xSuccess := __QUERYINTERFACE(iq_stExampleLeafModuleItf.i_ifDrive, ifRefActualValuesPosition);
IF NOT xSuccess OR ifRefActualValuesPosition = 0 THEN
	stExceptionModuleReaction1.etDiag		:= GD.ET_Diag.InputParameterInvalid;
	stExceptionModuleReaction1.udiDiagExt	:= ET_DiagExtExampleLeafModule.DriveInvalid;
	stExceptionModuleReaction1.sMsg			:= 'i_ifDrive : IF_RefActualValues not implemented.';
	
	ReportException(iq_stException := stExceptionModuleReaction1);		
END_IF
END_METHOD

METHOD SetOutputs
VAR_INPUT
END_VAR
IF xNotAbleToSetException THEN
	; (* Do nothing. Diag outputs show not reportable exception *)
	iq_stStandardModuleItf.q_xReady := FALSE;
ELSIF stModuleReaction.axReaction[TPL.ET_Reaction.AsyncStop] THEN
	iq_stStandardModuleItf.q_etDiag := GD.ET_Diag.ExecutionAborted;
	iq_stStandardModuleItf.q_udiDiagExt := ET_DiagExtExampleLeafModule.AsyncStop;
	iq_stStandardModuleItf.q_sDiagExt := 'AsyncStop';
	iq_stStandardModuleItf.q_sMsg := '';
	
	iq_stStandardModuleItf.q_xReady := FALSE;
ELSIF stModuleReaction.axReaction[TPL.ET_Reaction.SyncStopEL] THEN
	iq_stStandardModuleItf.q_etDiag := GD.ET_Diag.ExecutionAborted;
	iq_stStandardModuleItf.q_udiDiagExt := ET_DiagExtExampleLeafModule.SyncStopEL;
	iq_stStandardModuleItf.q_sDiagExt := 'SyncStopEL';
	iq_stStandardModuleItf.q_sMsg := '';
	
	iq_stStandardModuleItf.q_xReady := FALSE;
ELSIF stModuleReaction.axReaction[TPL.ET_Reaction.SyncStopEH] THEN
	iq_stStandardModuleItf.q_etDiag := GD.ET_Diag.ExecutionAborted;
	iq_stStandardModuleItf.q_udiDiagExt := ET_DiagExtExampleLeafModule.SyncStopEH;
	iq_stStandardModuleItf.q_sDiagExt := 'SyncStopEH';
	iq_stStandardModuleItf.q_sMsg := '';
	
	iq_stStandardModuleItf.q_xReady := FALSE;
ELSIF stModuleReaction.axReaction[TPL.ET_Reaction.StopEndOfCycle] THEN
	iq_stStandardModuleItf.q_etDiag := GD.ET_Diag.ExecutionAborted;
	iq_stStandardModuleItf.q_udiDiagExt := ET_DiagExtExampleLeafModule.StopEndOfCycle;
	iq_stStandardModuleItf.q_sDiagExt := 'StopEndOfCycle';
	iq_stStandardModuleItf.q_sMsg := '';
	
	iq_stStandardModuleItf.q_xReady := FALSE;
ELSE
	IF (iq_stExampleLeafModuleItf.q_etState <> ET_ExampleLeafModuleState.Disabled) AND
	   (iq_stExampleLeafModuleItf.q_etState <> ET_ExampleLeafModuleState.Initializing) THEN

		iq_stStandardModuleItf.q_xReady := TRUE;
	ELSE
		iq_stStandardModuleItf.q_xReady := FALSE;
	END_IF
		
	iq_stStandardModuleItf.q_etDiag := GD.ET_Diag.Ok;
	CASE iq_stExampleLeafModuleItf.q_etState OF
		ET_ExampleLeafModuleState.NoOp: 
			iq_stStandardModuleItf.q_udiDiagExt := ET_DiagExtExampleLeafModule.NoOp;
		ET_ExampleLeafModuleState.Disabled:
			iq_stStandardModuleItf.q_udiDiagExt := ET_DiagExtExampleLeafModule.Disabled;
		ET_ExampleLeafModuleState.Initializing:
			iq_stStandardModuleItf.q_udiDiagExt := ET_DiagExtExampleLeafModule.Initializing;
		ET_ExampleLeafModuleState.HomingWaitForStart:
			iq_stStandardModuleItf.q_udiDiagExt := ET_DiagExtExampleLeafModule.HomingWaitForStart;
		ET_ExampleLeafModuleState.HomingExecuting:
			iq_stStandardModuleItf.q_udiDiagExt := ET_DiagExtExampleLeafModule.HomingExecuting;
		ET_ExampleLeafModuleState.HomingDone:
			iq_stStandardModuleItf.q_udiDiagExt := ET_DiagExtExampleLeafModule.HomingDone;
		ET_ExampleLeafModuleState.AutoWaitForStart:
			iq_stStandardModuleItf.q_udiDiagExt := ET_DiagExtExampleLeafModule.AutoWaitForStart;
		ET_ExampleLeafModuleState.AutoRunning:
			iq_stStandardModuleItf.q_udiDiagExt := ET_DiagExtExampleLeafModule.AutoRunning;
	END_CASE
	iq_stStandardModuleItf.q_sDiagExt := FC_EtDiagExtExampleLeafModuleToString(i_etDiagExt := iq_stStandardModuleItf.q_udiDiagExt);
	iq_stStandardModuleItf.q_sMsg := '';
END_IF

IF fbLoggerPoint.etLogLevel >= APL.ET_LogLevel.StatusMessage THEN
	IF (iq_stExampleLeafModuleItf.q_etState <> etStateOld) THEN
		fbLoggerPoint.AddLogEntry(	i_etLogLevel	:= APL.ET_LogLevel.StatusMessage,
									i_etDiag		:= GD.ET_Diag.Ok,
									i_udiDiagExt	:= ET_DiagExtExampleLeafModule.Ok,
									i_sMessage		:= Standard.CONCAT('State changed to: ', FC_EtExampleLeafModuleStateToString(i_etState := iq_stExampleLeafModuleItf.q_etState)),
									q_etDiag		:= ,
									q_etDiagExt		:= );
	END_IF
	etStateOld := iq_stExampleLeafModuleItf.q_etState;
END_IF
END_METHOD

ACTION SignalSuccessfulExecution:
IF fbLoggerPoint.etLogLevel >= APL.ET_LogLevel.StatusMessage THEN
	fbLoggerPoint.AddLogEntry(	i_etLogLevel	:= APL.ET_LogLevel.StatusMessage,
								i_etDiag		:= GD.ET_Diag.Ok,
								i_udiDiagExt	:= ET_DiagExtExampleLeafModule.Ok,
								i_sMessage		:= Standard.CONCAT(Standard.CONCAT(Standard.CONCAT('Command done: ', FC_etExampleLeafModuleCmdToString(i_diCmd := iq_stStandardModuleItf.iq_diCmd)),' number: '),DINT_TO_STRING(iq_stStandardModuleItf.iq_diCmd)),
								q_etDiag		:= ,
								q_etDiagExt		:= );
END_IF

iq_stStandardModuleItf.q_xCMDActive := FALSE;
iq_stStandardModuleItf.q_xCMDDone := TRUE;
IF(iq_stStandardModuleItf.iq_diCMD = iq_stStandardModuleItf.q_diCMDActive) THEN
	iq_stStandardModuleItf.iq_diCMD := 0;
(* ELSE don't touch iq_diCMD *)
END_IF
END_ACTION

ACTION SignalUnSuccessfulExecution:
IF fbLoggerPoint.etLogLevel >= APL.ET_LogLevel.StatusMessage THEN
	fbLoggerPoint.AddLogEntry(	i_etLogLevel	:= APL.ET_LogLevel.StatusMessage,
								i_etDiag		:= GD.ET_Diag.Ok,
								i_udiDiagExt	:= ET_DiagExtExampleLeafModule.Ok,
								i_sMessage		:= Standard.CONCAT(Standard.CONCAT(Standard.CONCAT('Command failed: ', FC_etExampleLeafModuleCmdToString(i_diCmd := iq_stStandardModuleItf.iq_diCmd)),' number: '),DINT_TO_STRING(iq_stStandardModuleItf.iq_diCmd)),
								q_etDiag		:= ,
								q_etDiagExt		:= );
END_IF

iq_stStandardModuleItf.q_xCMDActive := FALSE;
iq_stStandardModuleItf.q_xCMDDone := FALSE;
IF(iq_stStandardModuleItf.iq_diCMD = iq_stStandardModuleItf.q_diCMDActive) THEN
	iq_stStandardModuleItf.iq_diCMD := - iq_stStandardModuleItf.iq_diCMD;
(* ELSE don't touch iq_diCMD *)
END_IF
END_ACTION

END_FUNCTION_BLOCK

// LMC_PacDrive/Application/TemplateFullProgrammingFramework/Examples/ExampleLeafModule/FC_EtExampleLeafModuleCmdToString
FUNCTION FC_EtExampleLeafModuleCmdToString : STRING[15]
VAR_INPUT
	i_diCmd		: DINT;
END_VAR
VAR_OUTPUT
	q_etDiag	: GD.ET_Diag := GD.ET_Diag.Ok;
	q_etDiagExt	: ET_DiagExtExampleLeafModule := ET_DiagExtExampleLeafModule.Ok;
END_VAR

CASE i_diCMD OF
	ET_ExampleLeafModuleCmd.Homing:
		FC_EtExampleLeafModuleCmdToString := 'Homing';
	ET_ExampleLeafModuleCmd.Auto:
		FC_EtExampleLeafModuleCmdToString := 'Auto';
	ET_ExampleLeafModuleCmd.Stop:
		FC_EtExampleLeafModuleCmdToString := 'Stop';
	ET_ExampleLeafModuleCmd.Start:
		FC_EtExampleLeafModuleCmdToString := 'Start';
	ET_ExampleLeafModuleCmd.Hold:
		FC_EtExampleLeafModuleCmdToString := 'Hold';
	ELSE
		FC_EtExampleLeafModuleCmdToString := CONCAT('Unkown Cmd ', DINT_TO_STRING(i_diCMD));
		
		q_etDiag := GD.ET_Diag.InputParameterInvalid;
		q_etDiagExt := ET_DiagExtExampleLeafModule.UnknownCmd;
END_CASE

END_FUNCTION

// LMC_PacDrive/Application/TemplateFullProgrammingFramework/Examples/ExampleLeafModule/FC_EtExampleLeafModuleStateToString
FUNCTION FC_EtExampleLeafModuleStateToString : STRING[25]
VAR_INPUT
	i_etState	: ET_ExampleLeafModuleState;
END_VAR
VAR_OUTPUT
	q_etDiag	: GD.ET_Diag := GD.ET_Diag.Ok;
	q_etDiagExt	: ET_DiagExtExampleLeafModule := ET_DiagExtExampleLeafModule.Ok;
END_VAR

CASE i_etState OF
	ET_ExampleLeafModuleState.Disabled:
		FC_EtExampleLeafModuleStateToString := 'Disabled';
	ET_ExampleLeafModuleState.Initializing:
		FC_EtExampleLeafModuleStateToString := 'Initializing';
	ET_ExampleLeafModuleState.NoOp:
		FC_EtExampleLeafModuleStateToString := 'NoOp';
	ET_ExampleLeafModuleState.HomingWaitForStart:
		FC_EtExampleLeafModuleStateToString := 'HomingWaitForStart';
	ET_ExampleLeafModuleState.HomingExecuting:
		FC_EtExampleLeafModuleStateToString := 'HomingExecuting';
	ET_ExampleLeafModuleState.HomingDone:
		FC_EtExampleLeafModuleStateToString := 'HomingDone';
	ET_ExampleLeafModuleState.AutoWaitForStart:
		FC_EtExampleLeafModuleStateToString := 'AutoWaitForStart';
	ET_ExampleLeafModuleState.AutoRunning:
		FC_EtExampleLeafModuleStateToString := 'AutoRunning';
	ELSE
		FC_EtExampleLeafModuleStateToString := CONCAT('Unkown State ', UDINT_TO_STRING(i_etState));
		
		q_etDiag := GD.ET_Diag.InputParameterInvalid;
		q_etDiagExt := ET_DiagExtExampleLeafModule.UnknownState;
END_CASE

END_FUNCTION

// LMC_PacDrive/Application/TemplateFullProgrammingFramework/Examples/ExampleLeafModule/FC_EtDiagExtExampleLeafModuleToString
FUNCTION FC_EtDiagExtExampleLeafModuleToString : STRING[80]

VAR_INPUT
	i_etDiagExt : ET_DiagExtExampleLeafModule;
END_VAR

VAR_OUTPUT
	q_etDiag	: GD.ET_Diag := GD.ET_Diag.Ok;
	q_etDiagExt	: ET_DiagExtExampleLeafModule := ET_DiagExtExampleLeafModule.Ok;
END_VAR

VAR
END_VAR

CASE i_etDiagExt OF
	ET_DiagExtExampleLeafModule.Ok:										FC_EtDiagExtExampleLeafModuleToString := 'Ok';
	ET_DiagExtExampleLeafModule.Disabled:								FC_EtDiagExtExampleLeafModuleToString := 'Disabled';
	ET_DiagExtExampleLeafModule.Initializing:							FC_EtDiagExtExampleLeafModuleToString := 'Initializing';
	ET_DiagExtExampleLeafModule.NoOp:									FC_EtDiagExtExampleLeafModuleToString := 'NoOp';
	ET_DiagExtExampleLeafModule.HomingWaitForStart:						FC_EtDiagExtExampleLeafModuleToString := 'HomingWaitForStart';
	ET_DiagExtExampleLeafModule.HomingExecuting:						FC_EtDiagExtExampleLeafModuleToString := 'HomingExecuting';
	ET_DiagExtExampleLeafModule.HomingDone:								FC_EtDiagExtExampleLeafModuleToString := 'HomingDone';
	ET_DiagExtExampleLeafModule.AutoWaitForStart:						FC_EtDiagExtExampleLeafModuleToString := 'AutoWaitForStart';
	ET_DiagExtExampleLeafModule.AutoRunning:							FC_EtDiagExtExampleLeafModuleToString := 'AutoRunning';
	ET_DiagExtExampleLeafModule.Working:								FC_EtDiagExtExampleLeafModuleToString := 'Working';

	ET_DiagExtExampleLeafModule.UnknownDiagExtExampleLeafModule:		FC_EtDiagExtExampleLeafModuleToString := 'UnknownDiagExtExampleLeafModule';
	ET_DiagExtExampleLeafModule.SubModuleAddInterfacesInvalidPointer:	FC_EtDiagExtExampleLeafModuleToString := 'SubModuleAddInterfacesInvalidPointer';
	ET_DiagExtExampleLeafModule.SubModuleConstantRange:					FC_EtDiagExtExampleLeafModuleToString := 'SubModuleConstantRange';
	ET_DiagExtExampleLeafModule.MissingExtInit:							FC_EtDiagExtExampleLeafModuleToString := 'MissingExtInit';
	ET_DiagExtExampleLeafModule.ReactionOffsetRange:					FC_EtDiagExtExampleLeafModuleToString := 'ReactionOffsetRange';
	ET_DiagExtExampleLeafModule.DriveInvalid:							FC_EtDiagExtExampleLeafModuleToString := 'DriveInvalid';
	
	ET_DiagExtExampleLeafModule.CmdUnknown:								FC_EtDiagExtExampleLeafModuleToString := 'CmdUnknown';
	ET_DiagExtExampleLeafModule.CmdImpossibleOverwrite:					FC_EtDiagExtExampleLeafModuleToString := 'CmdImpossibleOverwrite';
	ET_DiagExtExampleLeafModule.CmdImpossibleState:						FC_EtDiagExtExampleLeafModuleToString := 'CmdImpossibleState';
	ET_DiagExtExampleLeafModule.CmdImpossibleReaction:					FC_EtDiagExtExampleLeafModuleToString := 'CmdImpossibleReaction';
	
	ET_DiagExtExampleLeafModule.AsyncStop:								FC_EtDiagExtExampleLeafModuleToString := 'AsyncStop';
	ET_DiagExtExampleLeafModule.SyncStopEL:								FC_EtDiagExtExampleLeafModuleToString := 'SyncStopEL';
	ET_DiagExtExampleLeafModule.SyncStopEH:								FC_EtDiagExtExampleLeafModuleToString := 'SyncStopEH';
	ET_DiagExtExampleLeafModule.StopEndOfCycle:							FC_EtDiagExtExampleLeafModuleToString := 'StopEndOfCycle';
	
	ET_DiagExtExampleLeafModule.DriveFatalException:					FC_EtDiagExtExampleLeafModuleToString := 'DriveFatalException';
	ET_DiagExtExampleLeafModule.DriveException:							FC_EtDiagExtExampleLeafModuleToString := 'DriveException';
	ET_DiagExtExampleLeafModule.DriveWarning:							FC_EtDiagExtExampleLeafModuleToString := 'DriveWarning';
	
	ET_DiagExtExampleLeafModule.UnknownState:							FC_EtDiagExtExampleLeafModuleToString := 'UnknownState';
	ET_DiagExtExampleLeafModule.UnknownCmd:								FC_EtDiagExtExampleLeafModuleToString := 'UnknownCmd';
	ET_DiagExtExampleLeafModule.RandomException:						FC_EtDiagExtExampleLeafModuleToString := 'RandomException';

	ET_DiagExtExampleLeafModule.CurrentStandardItfInvalidPointer:		FC_EtDiagExtExampleLeafModuleToString := 'CurrentStandardItfInvalidPointer';
	ET_DiagExtExampleLeafModule.CurrentAddItfInvalidPointer:			FC_EtDiagExtExampleLeafModuleToString := 'CurrentAddItfInvalidPointer';
	
	ET_DiagExtExampleLeafModule.ParentInvalid:							FC_EtDiagExtExampleLeafModuleToString := 'ParentInvalid';
	ET_DiagExtExampleLeafModule.ParentNotRegistered:					FC_EtDiagExtExampleLeafModuleToString := 'ParentNotRegistered';
	ET_DiagExtExampleLeafModule.MaxNumberOfLoggerPointsExeeded:			FC_EtDiagExtExampleLeafModuleToString := 'MaxNumberOfLoggerPointsExeeded';
	ET_DiagExtExampleLeafModule.UnexpectedDiagExt:						FC_EtDiagExtExampleLeafModuleToString := 'UnexpectedDiagExt';
	
	ELSE
		FC_EtDiagExtExampleLeafModuleToString := Standard.CONCAT('Unkown ET_DiagExtExampleLeafModule ', UDINT_TO_STRING(i_etDiagExt));
		
		q_etDiag	:= GD.ET_Diag.InputParameterInvalid;
		q_etDiagExt	:= ET_DiagExtExampleLeafModule.UnknownDiagExtExampleLeafModule;
END_CASE

END_FUNCTION

// LMC_PacDrive/Application/TemplateFullProgrammingFramework/Examples/ExampleLeafModule/FB_ExampleLeafModuleController
FUNCTION_BLOCK FB_ExampleLeafModuleController

VAR_INPUT
	i_xEnable				: BOOL;
END_VAR

VAR_IN_OUT
	iq_stStandardModuleItf	: TPL.ST_StandardModuleInterface;
	iq_stStandardMotionItf	: TPL.ST_StandardMotionInterface;
	iq_stExceptionList		: TPL.ST_ExceptionList;
	iq_stLogDataList		: TPL.ST_LogDataList;
END_VAR

VAR_OUTPUT
	q_xActive				: BOOL;
	q_xReady				: BOOL;
	q_etDiag				: GD.ET_Diag := GD.ET_Diag.Ok;
	q_etDiagExt				: ET_DiagExtExampleLeafModule := ET_DiagExtExampleLeafModule.Disabled;
	q_sMsg					: STRING[80] := '';
END_VAR

VAR
	xEnableFlag				: BOOL;
	udiTmp					: UDINT;
END_VAR

IF i_xEnable AND NOT xEnableFlag THEN
	xEnableFlag	:= TRUE;
	
	q_xActive	:= TRUE;

	q_etDiag	:= GD.ET_Diag.Ok;
	q_etDiagExt := ET_DiagExtExampleLeafModule.Initializing;
	q_sMsg		:= '';
	
	IF ((iq_stStandardModuleItf.iq_stExt.udiNumberOfSubModules <> 0) AND 
	   ((iq_stStandardModuleItf.iq_stExt.pdwSubModulesAddItf = 0) OR (iq_stStandardModuleItf.iq_stExt.dwSubModulesItf = 0))) THEN
	   
		q_etDiag	:= GD.ET_Diag.ExecutionAborted;
		q_etDiagExt	:= ET_DiagExtExampleLeafModule.MissingExtInit;
		q_sMsg		:= 'Missing call of FC_UpdateExampleLeafModuleAddInterfaceStruct';

		RETURN;
	END_IF
	
	udiTmp := ET_ExceptionSource.ExampleLeafModule;
	
	q_xReady := TPL.FC_CheckSubModuleList(	i_dwModuleType		:= UDINT_TO_DWORD(ET_ModuleType.ExampleLeafModule),
											i_udiModuleId		:= iq_stStandardModuleItf.i_udiModuleId,
											i_sModuleName		:= iq_stStandardModuleItf.i_sModuleName,
											i_etSource			:= udiTmp (* Hack around compiler restrictions *),
											iq_stExt			:= iq_stStandardModuleItf.iq_stExt,
											iq_stExceptionList	:= iq_stExceptionList,
											iq_stLogDataList	:= iq_stLogDataList);
											
	IF NOT q_xReady THEN
		xEnableFlag := FALSE;
	END_IF

ELSIF NOT i_xEnable AND xEnableFlag THEN
	xEnableFlag	:= FALSE;
	
	(* No actions required, this simple module does not support jogging or any other things the XXXModuleController would have to handle *)
	q_xReady 	:= FALSE;
	q_xActive	:= FALSE;
	
	q_etDiag	:= GD.ET_Diag.Ok;
	q_etDiagExt	:= ET_DiagExtExampleLeafModule.Disabled;
	q_sMsg		:= '';
END_IF



IF q_xActive AND q_xReady THEN
	(* No actions required, this simple module does not support jogging or any other things the XXXModuleController would have to handle *)
	q_etDiag	:= GD.ET_Diag.Ok;
	q_etDiagExt := ET_DiagExtExampleLeafModule.Working;
	q_sMsg		:= '';
END_IF

END_FUNCTION_BLOCK

// LMC_PacDrive/Application/TemplateFullProgrammingFramework/Examples/ExampleLeafModule/FC_UpdateExampleLeafModuleAddInterfaceStruct
FUNCTION FC_UpdateExampleLeafModuleAddInterfaceStruct : BOOL

VAR_INPUT
	i_pdwSubModuleAddInterfaces		: POINTER TO DWORD;
	i_udiSubModuleConstant			: UDINT;
END_VAR

VAR_OUTPUT
	q_etDiag						: GD.ET_Diag := GD.ET_Diag.Ok;
	q_etDiagExt						: ET_DiagExtExampleLeafModule := ET_DiagExtExampleLeafModule.Ok;
	q_sMsg							: STRING[80] := '';
END_VAR

VAR_IN_OUT
	iq_stExampleLeafModuleInterface	: ST_ExampleLeafModuleInterface;
END_VAR

VAR
	pdwArrayPos						: POINTER TO DWORD;
END_VAR

IF i_pdwSubModuleAddInterfaces = 0 THEN
	q_etDiag	:= GD.ET_Diag.InputParameterInvalid;
	q_etDiagExt	:= ET_DiagExtExampleLeafModule.SubModuleAddInterfacesInvalidPointer;
	q_sMsg		:= '';
ELSIF i_udiSubModuleConstant < 1 THEN
	q_etDiag	:= GD.ET_Diag.InputParameterInvalid;
	q_etDiagExt := ET_DiagExtExampleLeafModule.SubModuleConstantRange;
	q_sMsg		:= '1 <= i_udiSubModuleConstant';
ELSE
	pdwArrayPos := i_pdwSubModuleAddInterfaces + UDINT_TO_DWORD((i_udiSubModuleConstant-1) * SIZEOF(pdwArrayPos^));
	pdwArrayPos^ := ADR(iq_stExampleLeafModuleInterface);
END_IF

END_FUNCTION

// LMC_PacDrive/Application/TemplateFullProgrammingFramework/EquipmentModules/MulticarrierModule/Multicarrier Stations/Test Multicarrier/FB_MotionTestStationBase
FUNCTION_BLOCK FB_MotionTestStationBase EXTENDS MCRS.FB_CoreStation 
VAR
	ifTargetStation 		: MCRS.IF_CoreStation;

	ifCarrier				 : MCR.IF_Carrier;

	etStationType 			  : ET_StationType;
	lrProcessPosInStation	  : LREAL;
	lrProcessGap			  : LREAL;

	lrMaxVelocity			: LREAL;
	lrMaxAcceleration		: LREAL;
	lrMaxDeceleration		: LREAL;
	lrMaxJerk				: LREAL;

	xError_loc				: BOOL;
	etResultSource_loc		: ET_ResultSource;
	udiEtResult_loc			: UDINT;
	sETResult_loc			: STRING(255);
	etResultStation_loc		: ET_ResultStation;
	etResultMCR_loc			: MCR.ET_Result;
	etResultMCRS_loc		: MCRS.ET_Result;
	sResultMsg_loc			: STRING(255);

	iState					: INT;
	xStationReadyForJob_loc	: BOOL;
	udiLoop					: UDINT;

	
END_VAR

END_FUNCTION_BLOCK

// LMC_PacDrive/Application/TemplateFullProgrammingFramework/Visualization/VIS_Main
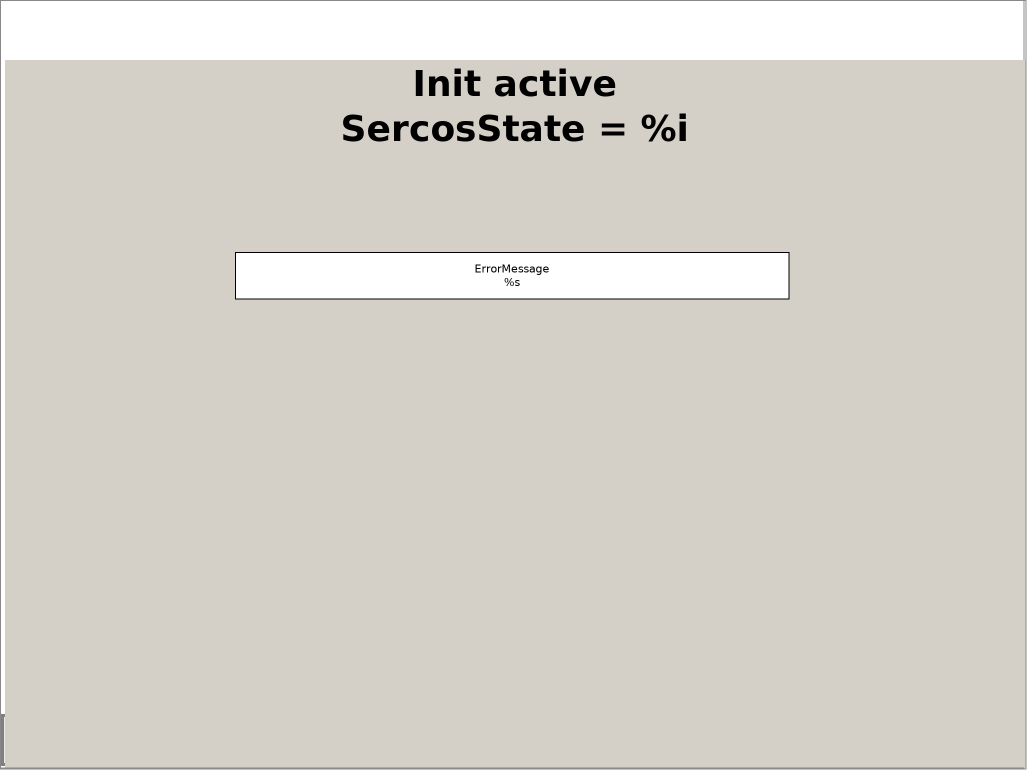
VISUALIZATION VIS_Main  // 1027x770
    Frame (0,0 1024x768)
        shows TPL.FR_NavControl1024x768(i_sTitle := 'Template: Main')
    Rectangle (105,63 688x480)
    Rectangle (105,63 688x40), "Machine - Control"
    Rectangle (105,102 688x78)
    Textfield (400,129 279x27)
    Button (693,119 90x44), "Diag Quit", colour toggle: SR_VisControl.vpq_xMachineInException
        p573394764: SR_VisControl.vpq_dwDiagQuitColor
        tap G_xDiagQuitEpas
    Textfield (117,129 279x27)
    Rectangle (402,130 275x25), "%s", text variable: SR_VisControl.vpq_etMainModuleControllerDiagExt, colour toggle: SR_VisControl.vpq_xMachineInException
        p2167032090: SR_VisControl.vpq_dwDiagQuitColor
    Rectangle (119,130 275x25), "%s", text variable: SR_VisControl.vpq_etMainModuleControllerDiag, colour toggle: SR_VisControl.vpq_xMachineInException
        p2167032090: SR_VisControl.vpq_dwDiagQuitColor
    Button (693,194 90x44), "Start", colour toggle: G_xStartEpas
        tap G_xStartEpas
    Button (693,253 90x44), "Stop", colour toggle: G_xStopEpas
        tap G_xStopEpas p3779583253=TRUE
    Button (693,312 90x44), "Jog +", colour toggle: G_xJogForwEpas
        tap G_xJogForwEpas p3779583253=TRUE
    Button (693,371 90x44), "Jog -", colour toggle: G_xJogBackEpas
        tap G_xJogBackEpas p3779583253=TRUE
    Button (125,195 90x44), "Prepare", colour toggle: G_xPrepareActive
        tap G_xDoPrepare
    Button (238,195 90x44), "Auto", colour toggle: G_xAutoActive
        tap G_xDoAuto
    Button (351,195 90x44), "Brake Release", colour toggle: G_xBrakeReleaseActive
        tap G_xDoBrakeRelease
    Button (464,195 90x44), "Jog Machine", colour toggle: G_xJogMachineActive
        tap G_xDoJogMachine
    Button (577,195 90x44), "Manual", colour toggle: G_xManualActive
        tap G_xDoManual
    Polyline (680,431) (793,431)
    Frame (693,442 90x90)
        shows TPL.FR_EmergencyStop90x90(i_xChangeColor := NOT G_xEmergencyEpas, i_xInvisible := FALSE, iq_xToggle := G_xEmergencyEpas)
    Frame (109,256 574x283)
        shows TPL.FR_ModuleCommandTable620x250(i_stCurrentModuleStandardItf := SR_VisControl.vpq_stMachineInterface, i_astActualCmdTable := SR_VisControl.vpq_astActualCmdTableMain, i_udiNumberOfCmdSteps := SR_VisControl.vpq_udiNumberOfCmdStepsMain, i_sCmdTitel := SR_VisControl.vpq_sCmdTitelMain, i_xDoEnable := SR_VisControl.vpq_xDoEnable, i_xDisableScrollUp := SR_VisControl.vpq_xDisableScrollUpMain, i_xDisableScrollDown := SR_VisControl.vpq_xDisableScrollDownMain, iq_udiIndexMin := SR_VisControl.vpiq_udiIndexMinMain)
        p2190627833: SR_VisControl.vpq_stMachineInterface
        p3492251336: SR_VisControl.vpq_stMachineInterface.iq_stExt.diActiveStep
    Frame (1,714 1024x54)
        shows FR_NavigationButtons()
    Rectangle (205,720 98x40), "Machine Control"
    Frame (821,60 200x430), invisible if: NOT SR_VisControl.vpiq_xShowControlFrame
        shows TPL.FR_MachineControl200x430(i_stMachineItf := SR_VisControl.vpq_stMachineInterface, i_xPrepareActive := G_xPrepareActive, i_xAutoActive := G_xAutoActive, i_xBrakeReleaseActive := G_xBrakeReleaseActive, i_xJogMachineActive := G_xJogMachineActive, i_xManualActive := G_xManualActive, i_xException := SR_VisControl.vpq_xMachineInException, i_dwDiagQuitColor := SR_VisControl.vpq_dwDiagQuitColor, iq_iPositionX := SR_VisControl.vpiq_iPositionX, iq_iPositionY := SR_VisControl.vpiq_iPositionY, iq_xEmergencyEpas := G_xEmergencyEpas, iq_xStartEpas := G_xStartEpas, iq_xStopEpas := G_xStopEpas, iq_xJogForwEpas := G_xJogForwEpas, iq_xJogBackEpas := G_xJogBackEpas, iq_xDoPrepare := G_xDoPrepare, iq_xDoAuto := G_xDoAuto, iq_xDoBrakeRelease := G_xDoBrakeRelease, iq_xDoJogMachine := G_xDoJogMachine, iq_xDoManual := G_xDoManual, iq_xDiagQuitEpas := G_xDiagQuitEpas)
        p1457045297: SR_VisControl.stMachineInterface.stQ.xError
        p1941967854: g_I_xEmergency_Epas
        p2531571229: g_I_xStart_Epas
        p1511842254: g_I_xStop_Epas
        p745511063: g_I_xJogForw_Epas
        p3518271027: g_I_xJogBack_Epas
        p1982879521: g_I_xErrorQuit_Epas
        p3866886353: SR_VisControl.dwErrorQuitColor
        p1761348311: SR_VisControl.vpq_stMachineInterface
        p3560616238: SR_VisControl.vpiq_iPositionX
        p2738717112: SR_VisControl.vpiq_iPositionY
    Rectangle (5,60 1020x707), "Init active SercosState = %i", text variable: G_ifSercos.State, invisible if: SR_MainMachine.xInitSuccessful
    Rectangle (235,252 554x47), "ErrorMessage %s", text variable: SR_MainMachine.stMachineInterface.q_sMsg, invisible if: SR_MainMachine.xInitSuccessful or not SR_MainMachine.xError
END_VISUALIZATION

// LMC_PacDrive/Application/TemplateFullProgrammingFramework/Visualization/Vis_Multicarrier
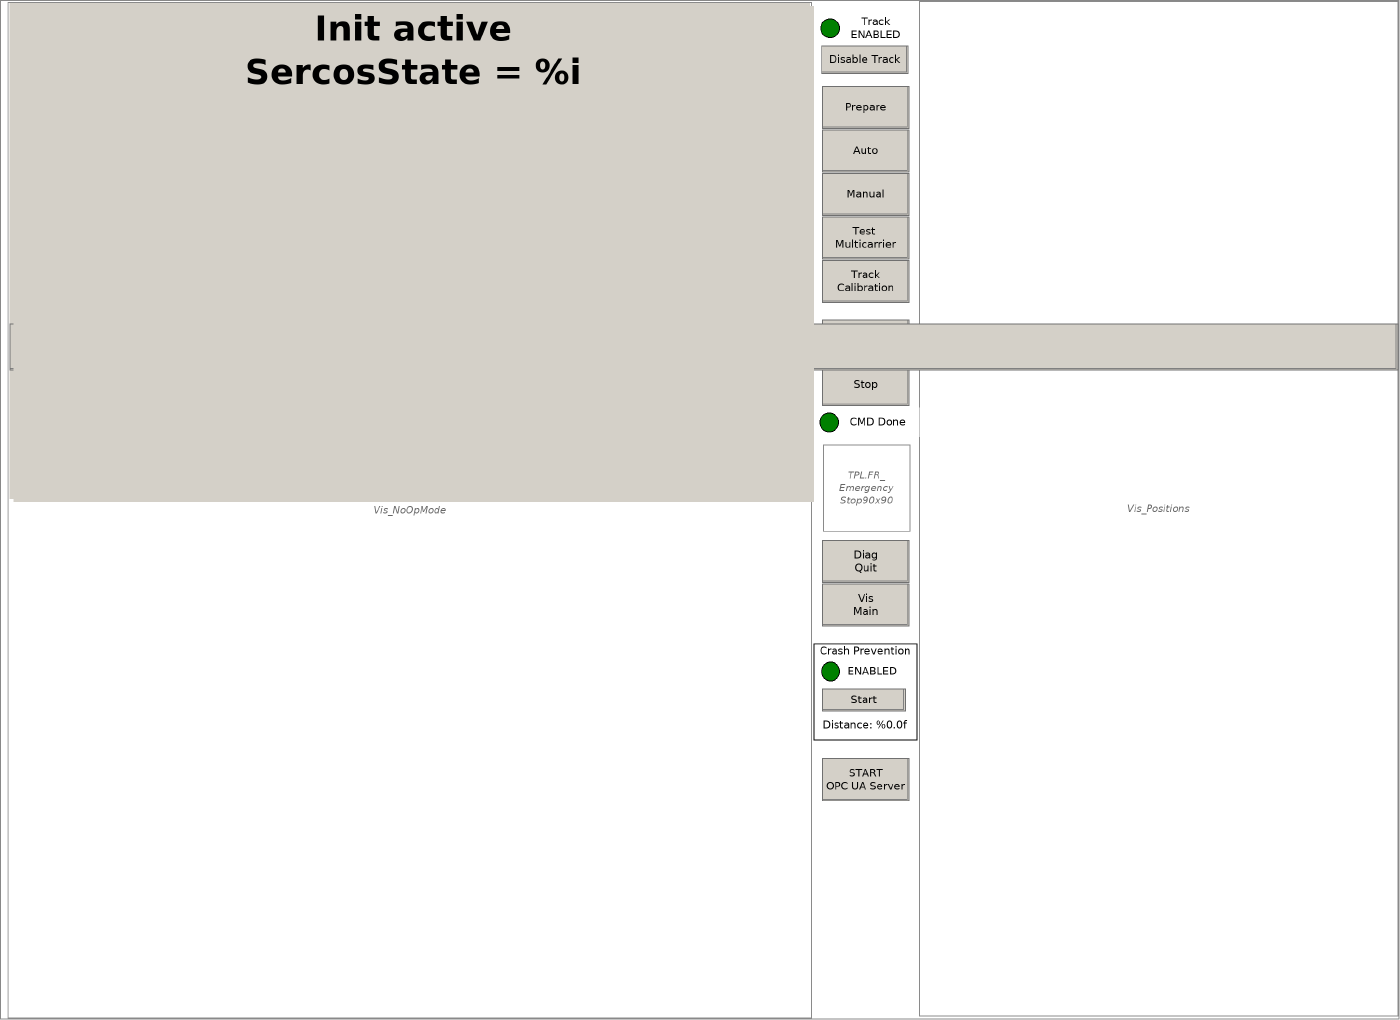
VISUALIZATION Vis_Multicarrier  // 1449x1056
    TabControl (8,2 832x1052), frame switch variable: SR_MultiCarrierModule.uiSetOpModeVis
        shows Vis_NoOpMode()
        shows Vis_Jogging()
        shows Vis_Auto()
        shows Vis_TestMulticarrier()
        shows Vis_TrackCalibration()
        [0]: TabTitle=None
        [1]: TabTitle=Manual
        [2]: TabTitle=Auto
        [3]: TabTitle=Test
        [4]: TabTitle=Trackcalibration
    TabControl (951,1 496x1051), frame switch variable: SR_MulticarrierModule.uiAdditionalVisTabs
        shows Vis_Positions()
        shows Vis_ApplicationLogger()
        shows Vis_Trace()
        shows Vis_Error()
        [0]: TabTitle=Positions
        [2]: TabTitle=Trace
        [3]: TabTitle=Error
    Frame (852,460 90x90)
        shows TPL.FR_EmergencyStop90x90(i_xChangeColor := NOT G_xEmergencyEpas, i_xInvisible := FALSE, iq_xToggle := G_xEmergencyEpas)
    Button (851,89 90x44), "Prepare", colour toggle: G_xPrepareActive
        tap G_xDoPrepare
    Button (851,559 90x44), "Diag Quit", colour toggle: SR_VisControl.vpq_xMachineInException
        p573394764: SR_VisControl.vpq_dwDiagQuitColor
        tap G_xDiagQuitEpas
    Button (851,134 90x44), "Auto", colour toggle: G_xAutoActive
        tap G_xDoAuto
    Button (851,179 90x44), "Manual", colour toggle: G_xManualActive
        tap G_xDoManual
    Button (851,224 90x44), "Test Multicarrier", colour toggle: G_xTestMulticarrierActive
        tap G_xDoTestMulticarrier
    Button (851,331 90x44), "Start", colour toggle: G_xStartEpas
        tap G_xStartEpas
    Button (851,376 90x44), "Stop", colour toggle: G_xStopEpas
        tap G_xStopEpas p3779583253=TRUE
    Button (851,785 90x44), "START OPC UA Server", colour toggle: SR_OpcUa.xStartUaServer
        toggle SR_OpcUa.xStartUaServer
    Group (848,422 103x30)
        Rectangle (18,0 85x30), "CMD Done"
        Ellipse (0,5 20x20), colour toggle: SR_MainMachine.fbModuleController.q_xCmdDone
    Rectangle (864,14 85x30), "Track ENABLED"
    Ellipse (849,19 20x20), colour toggle: SR_MultiCarrierModule.xEnableTrackSuccessful
    Button (850,47 90x29), "Enable Track", colour toggle: SR_MultiCarrierModule.xControlEnable, invisible if: SR_MultiCarrierModule.iStateOpMode > 0 or SR_MultiCarrierModule.xControlEnable
        toggle SR_MultiCarrierModule.xControlEnable
    Button (850,47 90x29), "Disable Track", invisible if: SR_MultiCarrierModule.iStateOpMode > 0 or not SR_MultiCarrierModule.xControlEnable
        toggle SR_MultiCarrierModule.xControlEnable
    Button (851,604 90x44), "Vis Main"
        OnMouseClick:  Assign=VIS_Main, Type=Assignment
    Rectangle (842,666 107x100), "Crash Prevention"
    Button (851,713 86x23), "Start", colour toggle: SR_MultiCarrierModule.xStartFbCrashPrevention
        toggle SR_MultiCarrierModule.xStartFbCrashPrevention
    Rectangle (863,680 80x30), "ENABLED"
    Ellipse (850,685 19x20), colour toggle: SR_MultiCarrierModule.xActiveFbCrashPrevention
    Rectangle (847,737 96x27), "Distance: %0.0f", tooltip "min distance between two Carriers (rear- and front offset under consideration)", text variable: GVL_Project.G_lrCrashDistance
        OnMouseClick: write the text variable via Default, min 0
    Rectangle (10,3 828x513), "Prepare Mode active", invisible if: SR_MulticarrierModule.iStateOpMode < 200 or SR_MulticarrierModule.iStateOpMode > 260
    Rectangle (149,192 554x47), "ErrorMessage %s", text variable: SR_MainMachine.stMachineInterface.q_sMsg, invisible if: SR_MainMachine.xInitSuccessful or not SR_MainMachine.xError
    Button (10,335 1437x48), "Enable Vis", colour toggle: G_xDoEnableVis, invisible if: G_xDoEnableVis
        toggle G_xDoEnableVis
    Rectangle (14,6 828x513), "Init active SercosState = %i", text variable: G_ifSercos.State, invisible if: SR_MainMachine.xInitSuccessful
    Button (851,269 90x44), "Track Calibration", colour toggle: G_xTrackCalibrationActive, invisible if: GVL_Project.Gc_xTrackCalibrationOfMulticarrier = false
        tap G_xDoTrackCalibration
END_VISUALIZATION

// LMC_PacDrive/Application/TemplateFullProgrammingFramework/Visualization/Examples/FR_ButtonAssignId
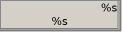
VISUALIZATION FR_ButtonAssignId  // 122x32
VAR_INPUT
	i_udiId : UDINT;
	i_sName : STRING[80];
	i_udiCurrentModuleId : UDINT;
END_VAR
VAR_IN_OUT
	iq_udiAssignTarget : UDINT;
END_VAR
    Button (0,0 120x30), "%s", text variable: i_sName, colour toggle: i_udiId = i_udiCurrentModuleId, invisible if: i_udiId<1
    Rectangle (0,0 119x29), "%s", text variable: i_udiId, invisible if: i_udiId<1
        OnMouseUp: execute { iq_udiAssignTarget := i_udiId; }
END_VISUALIZATION

// LMC_PacDrive/Application/TemplateFullProgrammingFramework/Visualization/Examples/FR_ExampleLeafModule
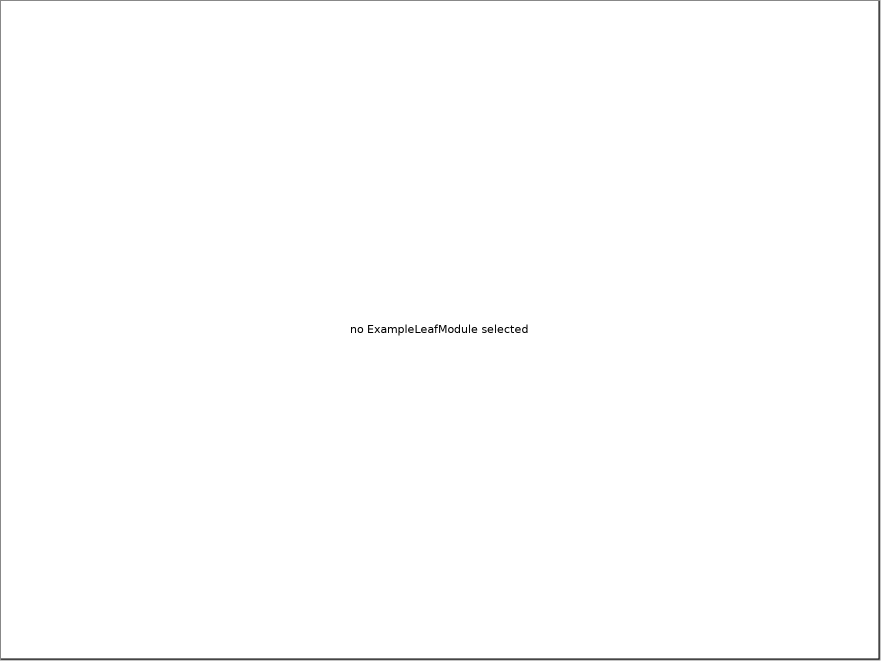
VISUALIZATION FR_ExampleLeafModule  // 881x661
VAR_IN_OUT
	iq_xModuleReactionDown				: BOOL;
	iq_xModuleReactionUp				: BOOL;
	iq_diStartStepToSet					: DINT;
	iq_diCmdToSet						: DINT;
	iq_xEnableModuleClicked				: BOOL;
	iq_xSetCmdClicked					: BOOL;
	iq_fbVisContExHandling				: TPL.FB_VisControllerExceptionHandling;
	iq_fbExampleLeafModuleVisController : FB_ExampleLeafModuleVisController;
END_VAR
VAR_INPUT
	i_stCurrentModuleStandardInterface : TPL.ST_StandardModuleInterface;
	i_sCurrentModuleReaction	: STRING[80];
	i_udiModuleReactionIndexMin : UDINT;
	i_axModuleReaction			: ARRAY [1..10] OF BOOL;
	i_udiNumberOfReactions 		: UDINT;
END_VAR
    Frame (0,0 380x211)
        shows TPL.FR_StandardModuleInterface380x220(i_stCurrentModuleStandardItf := i_stCurrentModuleStandardInterface, i_sCurrentModuleReaction := i_sCurrentModuleReaction, i_udiModuleReactionIndexMin := i_udiModuleReactionIndexMin, i_axModuleReaction := i_axModuleReaction, i_udiNumberOfReactions := i_udiNumberOfReactions, iq_xModuleReactionDown := iq_xModuleReactionDown, iq_xModuleReactionUp := iq_xModuleReactionUp, iq_diStartStepToSet := iq_diStartStepToSet, iq_diCmdToSet := iq_diCmdToSet, iq_xEnableModuleClicked := iq_xEnableModuleClicked, iq_xSetCmdClicked := iq_xSetCmdClicked, iq_fbVisContExHandling := iq_fbVisContExHandling)
        p3339340907: i_sZoomToVisModuleErrors
        p1094400588: i_xCurrentIsOfMyType
        p1029787830: i_fbVisContExHandling
        p2258115317: i_iModuleErrorReactionIndexMin
        p2777435286: i_axModuleErrorReaction
        p214250784: i_diNumberOfErrorreactions
        p311732222: iq_stCurrentModuleStandardInterface
        p640132070: iq_xModuleErrorReactionDown
        p4234372197: iq_xModuleErrorReactionUp
        p2938682392: iq_xEnableModule_Clicked
        p3592490199: iq_xSetCmd_Clicked
        p2307280719: iq_stCurrentModuleStandardInterface
        p2190627833: i_stCurrentModuleStandardInterface
    Rectangle (0,0 879x659), "no ExampleLeafModule selected", invisible if: iq_fbExampleLeafModuleVisController.xCurrentIsOfMyType
END_VISUALIZATION

// LMC_PacDrive/Application/TemplateFullProgrammingFramework/Visualization/Examples/FR_ExampleLeafModuleSelect
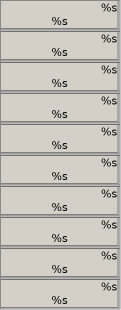
VISUALIZATION FR_ExampleLeafModuleSelect  // 121x310
VAR_IN_OUT
	iq_fbExampleLeafModuleVisController : FB_ExampleLeafModuleVisController;
END_VAR
VAR_INPUT
	i_stCurrentModuleStandardInterface : TPL.ST_StandardModuleInterface;
END_VAR
    Frame (0,0 119x29)
        shows FR_ButtonAssignId(i_udiId := iq_fbExampleLeafModuleVisController.audiExampleLeafModuleId[1], i_sName := iq_fbExampleLeafModuleVisController.asExampleLeafModuleName[1], i_udiCurrentModuleId := i_stCurrentModuleStandardInterface.i_udiModuleId, iq_udiAssignTarget := iq_fbExampleLeafModuleVisController.udiSetAsCurrentModule)
    Frame (0,31 119x29)
        shows FR_ButtonAssignId(i_udiId := iq_fbExampleLeafModuleVisController.audiExampleLeafModuleId[2], i_sName := iq_fbExampleLeafModuleVisController.asExampleLeafModuleName[2], i_udiCurrentModuleId := i_stCurrentModuleStandardInterface.i_udiModuleId, iq_udiAssignTarget := iq_fbExampleLeafModuleVisController.udiSetAsCurrentModule)
    Frame (0,62 119x29)
        shows FR_ButtonAssignId(i_udiId := iq_fbExampleLeafModuleVisController.audiExampleLeafModuleId[3], i_sName := iq_fbExampleLeafModuleVisController.asExampleLeafModuleName[3], i_udiCurrentModuleId := i_stCurrentModuleStandardInterface.i_udiModuleId, iq_udiAssignTarget := iq_fbExampleLeafModuleVisController.udiSetAsCurrentModule)
    Frame (0,93 119x29)
        shows FR_ButtonAssignId(i_udiId := iq_fbExampleLeafModuleVisController.audiExampleLeafModuleId[4], i_sName := iq_fbExampleLeafModuleVisController.asExampleLeafModuleName[4], i_udiCurrentModuleId := i_stCurrentModuleStandardInterface.i_udiModuleId, iq_udiAssignTarget := iq_fbExampleLeafModuleVisController.udiSetAsCurrentModule)
    Frame (0,124 119x29)
        shows FR_ButtonAssignId(i_udiId := iq_fbExampleLeafModuleVisController.audiExampleLeafModuleId[5], i_sName := iq_fbExampleLeafModuleVisController.asExampleLeafModuleName[5], i_udiCurrentModuleId := i_stCurrentModuleStandardInterface.i_udiModuleId, iq_udiAssignTarget := iq_fbExampleLeafModuleVisController.udiSetAsCurrentModule)
    Frame (0,155 119x29)
        shows FR_ButtonAssignId(i_udiId := iq_fbExampleLeafModuleVisController.audiExampleLeafModuleId[6], i_sName := iq_fbExampleLeafModuleVisController.asExampleLeafModuleName[6], i_udiCurrentModuleId := i_stCurrentModuleStandardInterface.i_udiModuleId, iq_udiAssignTarget := iq_fbExampleLeafModuleVisController.udiSetAsCurrentModule)
    Frame (0,186 119x29)
        shows FR_ButtonAssignId(i_udiId := iq_fbExampleLeafModuleVisController.audiExampleLeafModuleId[7], i_sName := iq_fbExampleLeafModuleVisController.asExampleLeafModuleName[7], i_udiCurrentModuleId := i_stCurrentModuleStandardInterface.i_udiModuleId, iq_udiAssignTarget := iq_fbExampleLeafModuleVisController.udiSetAsCurrentModule)
    Frame (0,217 119x29)
        shows FR_ButtonAssignId(i_udiId := iq_fbExampleLeafModuleVisController.audiExampleLeafModuleId[8], i_sName := iq_fbExampleLeafModuleVisController.asExampleLeafModuleName[8], i_udiCurrentModuleId := i_stCurrentModuleStandardInterface.i_udiModuleId, iq_udiAssignTarget := iq_fbExampleLeafModuleVisController.udiSetAsCurrentModule)
    Frame (0,248 119x29)
        shows FR_ButtonAssignId(i_udiId := iq_fbExampleLeafModuleVisController.audiExampleLeafModuleId[9], i_sName := iq_fbExampleLeafModuleVisController.asExampleLeafModuleName[9], i_udiCurrentModuleId := i_stCurrentModuleStandardInterface.i_udiModuleId, iq_udiAssignTarget := iq_fbExampleLeafModuleVisController.udiSetAsCurrentModule)
    Frame (0,279 119x29)
        shows FR_ButtonAssignId(i_udiId := iq_fbExampleLeafModuleVisController.audiExampleLeafModuleId[10], i_sName := iq_fbExampleLeafModuleVisController.asExampleLeafModuleName[10], i_udiCurrentModuleId := i_stCurrentModuleStandardInterface.i_udiModuleId, iq_udiAssignTarget := iq_fbExampleLeafModuleVisController.udiSetAsCurrentModule)
END_VISUALIZATION

// LMC_PacDrive/Application/TemplateFullProgrammingFramework/Visualization/Examples/VIS_ExampleLeafModule
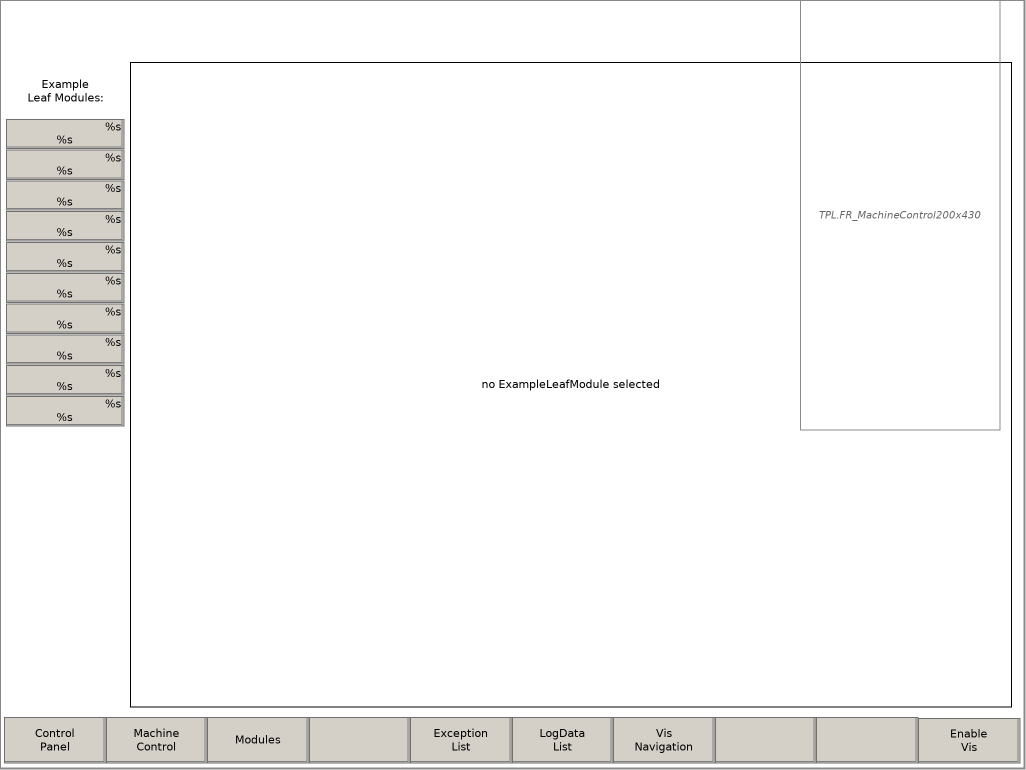
VISUALIZATION VIS_ExampleLeafModule  // 1026x770
    Frame (0,0 1024x768)
        shows TPL.FR_Nav1024x768(i_sTitle := 'Example Leaf Module')
    Frame (6,119 119x308)
        shows FR_ExampleLeafModuleSelect(i_stCurrentModuleStandardInterface := SR_VisControl.vpq_stCurrentModuleStandardInterface, iq_fbExampleLeafModuleVisController := SR_VisControl.vpiq_fbExampleLeafModuleVisController)
    Rectangle (6,65 119x52), "Example Leaf Modules:"
    Frame (130,62 884x647)
        shows FR_ExampleLeafModule(i_stCurrentModuleStandardInterface := SR_VisControl.vpq_stCurrentModuleStandardInterface, i_sCurrentModuleReaction := SR_VisControl.vpq_sCurrentModuleReaction, i_udiModuleReactionIndexMin := SR_VisControl.vpq_udiModuleReactionIndexMin, i_axModuleReaction := SR_VisControl.vpq_axModuleReaction, i_udiNumberOfReactions := TPL.Gc_udiMaxNumberOfReactions, iq_xModuleReactionDown := SR_VisControl.vpiq_xModuleReactionDown, iq_xModuleReactionUp := SR_VisControl.vpiq_xModuleReactionUp, iq_diStartStepToSet := SR_VisControl.vpiq_diStartStepToSet, iq_diCmdToSet := SR_VisControl.vpiq_diCmdToSet, iq_xEnableModuleClicked := SR_VisControl.vpiq_xEnableModuleClicked, iq_xSetCmdClicked := SR_VisControl.vpiq_xSetCmdClicked, iq_fbVisContExHandling := SR_VisControl.vpiq_fbVisContExHandling, iq_fbExampleLeafModuleVisController := SR_VisControl.vpiq_fbExampleLeafModuleVisController)
    Button (4,717 102x46), "Control Panel", colour toggle: SR_VisControl.vpiq_xShowControlFrame
        toggle SR_VisControl.vpiq_xShowControlFrame
    Button (106,717 101x46), "Machine Control"
        OnMouseClick:  Assign=VIS_Main, Type=Assignment
    Button (207,717 102x46), "Modules"
        OnMouseClick:  Assign=VIS_Modules, Type=Assignment
    Button (309,717 101x46)
    Button (410,717 102x46), "Exception List"
        OnMouseClick:  Assign=VIS_ExceptionList, Type=Assignment
    Button (512,717 101x46), "LogData List"
        OnMouseClick:  Assign=VIS_LogDataList, Type=Assignment
    Button (613,717 102x46), "Vis Navigation"
        OnMouseClick:  Assign=VIS_VisNavigation, Type=Assignment
    Button (715,717 101x46)
    Button (816,717 102x46)
    Button (918,718 102x45), "Enable Vis", colour toggle: G_xDoEnableVis
        OnMouseClick:  ToggleVariable=G_xDoEnableVis
    Frame (800,0 200x430), invisible if: NOT SR_VisControl.vpiq_xShowControlFrame
        shows TPL.FR_MachineControl200x430(i_stMachineItf := SR_VisControl.vpq_stMachineInterface, i_xPrepareActive := G_xPrepareActive, i_xAutoActive := G_xAutoActive, i_xBrakeReleaseActive := G_xBrakeReleaseActive, i_xJogMachineActive := G_xJogMachineActive, i_xManualActive := G_xManualActive, i_xException := SR_VisControl.vpq_xMachineInException, i_dwDiagQuitColor := SR_VisControl.vpq_dwDiagQuitColor, iq_iPositionX := SR_VisControl.vpiq_iPositionX, iq_iPositionY := SR_VisControl.vpiq_iPositionY, iq_xEmergencyEpas := G_xEmergencyEpas, iq_xStartEpas := G_xStartEpas, iq_xStopEpas := G_xStopEpas, iq_xJogForwEpas := G_xJogForwEpas, iq_xJogBackEpas := G_xJogBackEpas, iq_xDoPrepare := G_xDoPrepare, iq_xDoAuto := G_xDoAuto, iq_xDoBrakeRelease := G_xDoBrakeRelease, iq_xDoJogMachine := G_xDoJogMachine, iq_xDoManual := G_xDoManual, iq_xDiagQuitEpas := G_xDiagQuitEpas)
        p1457045297: SR_VisControl.stMachineInterface.stQ.xError
        p1941967854: g_I_xEmergency_Epas
        p2531571229: g_I_xStart_Epas
        p1511842254: g_I_xStop_Epas
        p745511063: g_I_xJogForw_Epas
        p3518271027: g_I_xJogBack_Epas
        p1982879521: g_I_xErrorQuit_Epas
        p3866886353: SR_VisControl.dwErrorQuitColor
        p1761348311: SR_VisControl.vpq_stMachineInterface
        p3560616238: SR_VisControl.vpiq_iPositionX - 800
        p2738717112: SR_VisControl.vpiq_iPositionY
END_VISUALIZATION

// LMC_PacDrive/Application/TemplateFullProgrammingFramework/Visualization/FramesProject/FR_ControlModuleTypes
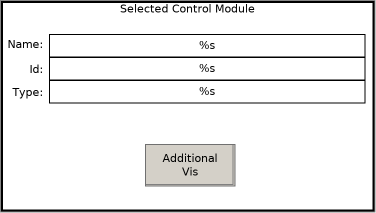
VISUALIZATION FR_ControlModuleTypes  // 376x213
VAR_INPUT
	i_sControlModuleName		: STRING[80];
	i_diControlModuleNumber		: DINT;
	i_diControlModuleType		: DINT;
END_VAR
    Rectangle (1,1 373x210), "Selected Control Module"
    Button (145,144 90x42), "Additional Vis"
        OnMouseClick:  AssignExpr=i_sZoomToControlModuleVis, Assign=VIS_ControlModule, Type=Assignment
    Textfield (49,34 316x23), "%s", text variable: i_sControlModuleName
    Rectangle (7,36 39x17), "Name:"
    Textfield (49,57 316x23), "%s", text variable: i_diControlModuleNumber
    Rectangle (7,61 39x17), "Id:"
    Rectangle (7,84 39x17), "Type:"
    Textfield (49,80 316x23), "%s", text variable: i_diControlModuleType
END_VISUALIZATION

// LMC_PacDrive/Application/TemplateFullProgrammingFramework/Visualization/FramesProject/FR_NavigationButtons
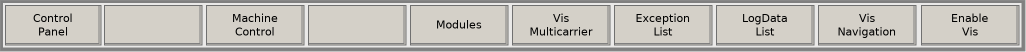
VISUALIZATION FR_NavigationButtons  // 1026x52
    Rectangle (0,0 1024x50)
    Button (410,5 98x40), "Modules"
        OnMouseClick:  Assign=VIS_Modules, Type=Assignment
    Button (5,5 96x40), "Control Panel", colour toggle: SR_VisControl.vpiq_xShowControlFrame
        toggle SR_VisControl.vpiq_xShowControlFrame
    Button (614,5 98x40), "Exception List"
        OnMouseClick:  Assign=VIS_ExceptionList, Type=Assignment
    Button (716,5 98x40), "LogData List"
        OnMouseClick:  Assign=VIS_LogDataList, Type=Assignment
    Button (818,5 98x40), "Vis Navigation"
        OnMouseClick:  Assign=VIS_VisNavigation, Type=Assignment
    Button (308,5 98x40)
    Button (104,5 98x40)
    Button (206,5 98x40), "Machine Control"
        OnMouseClick:  Assign=VIS_Main, Type=Assignment
    Button (921,5 98x40), "Enable Vis", colour toggle: G_xDoEnableVis
        toggle G_xDoEnableVis
    Button (512,5 98x40), "Vis Multicarrier"
        OnMouseDown:  Assign=Vis_Multicarrier, Type=Assignment
END_VISUALIZATION

// LMC_PacDrive/Application/TemplateFullProgrammingFramework/Visualization/FramesProject/FR_OtherModuleTypes
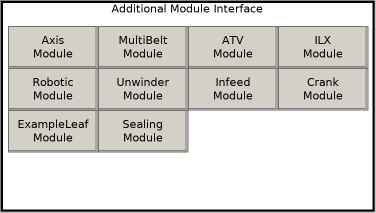
VISUALIZATION FR_OtherModuleTypes  // 376x213
    Rectangle (1,1 373x210), "Additional Module Interface"
    Button (8,26 90x42), "Axis Module", invisible if: SR_VisControl.vpq_stCurrentModuleStandardInterface.q_dwModuleType <> 3
        OnMouseClick:  Assign=VIS_AxisModule, Type=Assignment
    Button (98,26 90x42), "MultiBelt Module", invisible if: SR_VisControl.vpq_stCurrentModuleStandardInterface.q_dwModuleType <> 4
    Button (188,26 90x42), "ATV Module", invisible if: SR_VisControl.vpq_stCurrentModuleStandardInterface.q_dwModuleType <> 9
    Button (278,26 90x42), "ILX Module", invisible if: SR_VisControl.vpq_stCurrentModuleStandardInterface.q_dwModuleType <> 10
    Button (8,68 90x42), "Robotic Module", invisible if: SR_VisControl.vpq_stCurrentModuleStandardInterface.q_dwModuleType <> 6
    Button (8,110 90x42), "ExampleLeaf Module", invisible if: SR_VisControl.vpq_stCurrentModuleStandardInterface.q_dwModuleType <> 15000
        OnMouseClick:  AssignExpr=i_sZoomToExampleLeafModule, Assign=VIS_ExampleLeafModules, Type=Assignment
    Button (98,68 90x42), "Unwinder Module", invisible if: SR_VisControl.vpq_stCurrentModuleStandardInterface.q_dwModuleType <> 7
    Button (188,68 90x42), "Infeed Module", invisible if: SR_VisControl.vpq_stCurrentModuleStandardInterface.q_dwModuleType <> 5
    Button (278,68 90x42), "Crank Module", invisible if: SR_VisControl.vpq_stCurrentModuleStandardInterface.q_dwModuleType <> 11
    Button (98,110 90x42), "Sealing Module", invisible if: SR_VisControl.vpq_stCurrentModuleStandardInterface.q_dwModuleType <> 8
END_VISUALIZATION

// LMC_PacDrive/Application/TemplateFullProgrammingFramework/Visualization/Multicarrier/FR_CarDist
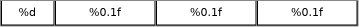
VISUALIZATION FR_CarDist  // 359x27
VAR_IN_OUT
	i_ifCarrierFeedback : MCR.IF_CarrierFeedback;
END_VAR
    Rectangle (1,0 53x25), "%d", text variable: i_ifCarrierFeedback.udiCarrierIndex
    Rectangle (55,0 100x25), "%0.1f", text variable: i_ifCarrierFeedback.ifFeedbackMotionValues.lrRefPosition
    Rectangle (156,0 100x25), "%0.1f", text variable: i_ifCarrierFeedback.ifFeedbackMotionValues.lrRefPosition
    Rectangle (257,0 100x25), "%0.1f", text variable: i_ifCarrierFeedback.ifFeedbackMotionValues.lrRefPosition
    Rectangle (55,0 100x25), "%0.1f", text variable: i_ifCarrierFeedback.ifFeedbackMotionValues.lrRefTrackPosition, invisible if: SR_MulticarrierModule.etVisPosColumn1 <> ET_VisPosGapDist.RefTrackPosition
    Rectangle (55,0 100x25), "%0.1f", text variable: i_ifCarrierFeedback.ifFeedbackToInFront.lrGapToCarrierInFront, invisible if: SR_MulticarrierModule.etVisPosColumn1 <> ET_VisPosGapDist.GapToCarrierInFront
    Rectangle (55,0 100x25), "%0.1f", text variable: i_ifCarrierFeedback.ifFeedbackToInFront.lrDistanceToCarrierInFront, invisible if: SR_MulticarrierModule.etVisPosColumn1 <> ET_VisPosGapDist.DistanceToCarrierInFront
    Rectangle (55,0 100x25), "%0.1f", text variable: i_ifCarrierFeedback.ifFeedbackToBehind.lrGapToCarrierBehind, invisible if: SR_MulticarrierModule.etVisPosColumn1 <> ET_VisPosGapDist.GapToCarrierBehind
    Rectangle (55,0 100x25), "%0.1f", text variable: i_ifCarrierFeedback.ifFeedbackToBehind.lrDistanceToCarrierBehind, invisible if: SR_MulticarrierModule.etVisPosColumn1 <> ET_VisPosGapDist.DistanceToCarrierBehind
    Rectangle (156,0 100x25), "%0.1f", text variable: i_ifCarrierFeedback.ifFeedbackMotionValues.lrRefTrackPosition, invisible if: SR_MulticarrierModule.etVisPosColumn2 <> ET_VisPosGapDist.RefTrackPosition
    Rectangle (156,0 100x25), "%0.1f", text variable: i_ifCarrierFeedback.ifFeedbackToInFront.lrGapToCarrierInFront, invisible if: SR_MulticarrierModule.etVisPosColumn2 <> ET_VisPosGapDist.GapToCarrierInFront
    Rectangle (156,0 100x25), "%0.1f", text variable: i_ifCarrierFeedback.ifFeedbackToInFront.lrDistanceToCarrierInFront, invisible if: SR_MulticarrierModule.etVisPosColumn2 <> ET_VisPosGapDist.DistanceToCarrierInFront
    Rectangle (156,0 100x25), "%0.1f", text variable: i_ifCarrierFeedback.ifFeedbackToBehind.lrGapToCarrierBehind, invisible if: SR_MulticarrierModule.etVisPosColumn2 <> ET_VisPosGapDist.GapToCarrierBehind
    Rectangle (156,0 100x25), "%0.1f", text variable: i_ifCarrierFeedback.ifFeedbackToBehind.lrDistanceToCarrierBehind, invisible if: SR_MulticarrierModule.etVisPosColumn2 <> ET_VisPosGapDist.DistanceToCarrierBehind
    Rectangle (257,0 100x25), "%0.1f", text variable: i_ifCarrierFeedback.ifFeedbackMotionValues.lrRefTrackPosition, invisible if: SR_MulticarrierModule.etVisPosColumn3 <> ET_VisPosGapDist.RefTrackPosition
    Rectangle (257,0 100x25), "%0.1f", text variable: i_ifCarrierFeedback.ifFeedbackToInFront.lrGapToCarrierInFront, invisible if: SR_MulticarrierModule.etVisPosColumn3 <> ET_VisPosGapDist.GapToCarrierInFront
    Rectangle (257,0 100x25), "%0.1f", text variable: i_ifCarrierFeedback.ifFeedbackToInFront.lrDistanceToCarrierInFront, invisible if: SR_MulticarrierModule.etVisPosColumn3 <> ET_VisPosGapDist.DistanceToCarrierInFront
    Rectangle (257,0 100x25), "%0.1f", text variable: i_ifCarrierFeedback.ifFeedbackToBehind.lrGapToCarrierBehind, invisible if: SR_MulticarrierModule.etVisPosColumn3 <> ET_VisPosGapDist.GapToCarrierBehind
    Rectangle (257,0 100x25), "%0.1f", text variable: i_ifCarrierFeedback.ifFeedbackToBehind.lrDistanceToCarrierBehind, invisible if: SR_MulticarrierModule.etVisPosColumn3 <> ET_VisPosGapDist.DistanceToCarrierBehind
END_VISUALIZATION

// LMC_PacDrive/Application/TemplateFullProgrammingFramework/Visualization/Multicarrier/FR_List
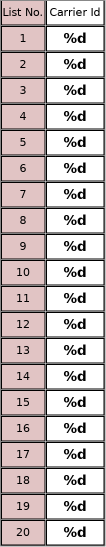
VISUALIZATION FR_List  // 106x547
VAR_IN_OUT
	iq_uiCarrierIndex :  ARRAY [1..MCR.GPL.Gc_udiMaxNumberOfCarriers] OF UDINT;
END_VAR
    Rectangle (46,26 58x25), "%d", text variable: iq_uiCarrierIndex[1], invisible if: iq_uiCarrierIndex[1] = 0
    Rectangle (1,26 44x25), "1", invisible if: iq_uiCarrierIndex[1] = 0
    Rectangle (46,52 58x25), "%d", text variable: iq_uiCarrierIndex[2], invisible if: iq_uiCarrierIndex[2] = 0
    Rectangle (1,52 44x25), "2", invisible if: iq_uiCarrierIndex[2] = 0
    Rectangle (46,78 58x25), "%d", text variable: iq_uiCarrierIndex[3], invisible if: iq_uiCarrierIndex[3] = 0
    Rectangle (1,78 44x25), "3", invisible if: iq_uiCarrierIndex[3] = 0
    Rectangle (46,104 58x25), "%d", text variable: iq_uiCarrierIndex[4], invisible if: iq_uiCarrierIndex[4] = 0
    Rectangle (1,104 44x25), "4", invisible if: iq_uiCarrierIndex[4] = 0
    Rectangle (46,130 58x25), "%d", text variable: iq_uiCarrierIndex[5], invisible if: iq_uiCarrierIndex[5] = 0
    Rectangle (1,130 44x25), "5", invisible if: iq_uiCarrierIndex[5] = 0
    Rectangle (46,156 58x25), "%d", text variable: iq_uiCarrierIndex[6], invisible if: iq_uiCarrierIndex[6] = 0
    Rectangle (1,156 44x25), "6", invisible if: iq_uiCarrierIndex[6] = 0
    Rectangle (46,182 58x25), "%d", text variable: iq_uiCarrierIndex[7], invisible if: iq_uiCarrierIndex[7] = 0
    Rectangle (1,182 44x25), "7", invisible if: iq_uiCarrierIndex[7] = 0
    Rectangle (46,0 58x25), "Carrier Id"
        OnMouseClick: write the text variable via Default
    Rectangle (1,0 44x25), "List No."
    Rectangle (46,208 58x25), "%d", text variable: iq_uiCarrierIndex[8], invisible if: iq_uiCarrierIndex[8] = 0
    Rectangle (1,208 44x25), "8", invisible if: iq_uiCarrierIndex[8] = 0
    Rectangle (46,234 58x25), "%d", text variable: iq_uiCarrierIndex[9], invisible if: iq_uiCarrierIndex[9] = 0
    Rectangle (1,234 44x25), "9", invisible if: iq_uiCarrierIndex[9] = 0
    Rectangle (46,260 58x25), "%d", text variable: iq_uiCarrierIndex[10], invisible if: iq_uiCarrierIndex[10] = 0
    Rectangle (1,260 44x25), "10", invisible if: iq_uiCarrierIndex[10] = 0
    Rectangle (46,286 58x25), "%d", text variable: iq_uiCarrierIndex[11], invisible if: iq_uiCarrierIndex[11] = 0
    Rectangle (1,286 44x25), "11", invisible if: iq_uiCarrierIndex[11] = 0
    Rectangle (46,312 58x25), "%d", text variable: iq_uiCarrierIndex[12], invisible if: iq_uiCarrierIndex[12] = 0
    Rectangle (1,312 44x25), "12", invisible if: iq_uiCarrierIndex[12] = 0
    Rectangle (46,338 58x25), "%d", text variable: iq_uiCarrierIndex[13], invisible if: iq_uiCarrierIndex[13] = 0
    Rectangle (1,338 44x25), "13", invisible if: iq_uiCarrierIndex[13] = 0
    Rectangle (46,364 58x25), "%d", text variable: iq_uiCarrierIndex[14], invisible if: iq_uiCarrierIndex[14] = 0
    Rectangle (1,364 44x25), "14", invisible if: iq_uiCarrierIndex[14] = 0
    Rectangle (46,390 58x25), "%d", text variable: iq_uiCarrierIndex[15], invisible if: iq_uiCarrierIndex[15] = 0
    Rectangle (1,390 44x25), "15", invisible if: iq_uiCarrierIndex[15] = 0
    Rectangle (46,416 58x25), "%d", text variable: iq_uiCarrierIndex[16], invisible if: iq_uiCarrierIndex[16] = 0
    Rectangle (1,416 44x25), "16", invisible if: iq_uiCarrierIndex[16] = 0
    Rectangle (46,442 58x25), "%d", text variable: iq_uiCarrierIndex[17], invisible if: iq_uiCarrierIndex[17] = 0
    Rectangle (1,442 44x25), "17", invisible if: iq_uiCarrierIndex[17] = 0
    Rectangle (46,468 58x25), "%d", text variable: iq_uiCarrierIndex[18], invisible if: iq_uiCarrierIndex[18] = 0
    Rectangle (1,468 44x25), "18", invisible if: iq_uiCarrierIndex[18] = 0
    Rectangle (46,494 58x25), "%d", text variable: iq_uiCarrierIndex[19], invisible if: iq_uiCarrierIndex[19] = 0
    Rectangle (1,494 44x25), "19", invisible if: iq_uiCarrierIndex[19] = 0
    Rectangle (46,520 58x25), "%d", text variable: iq_uiCarrierIndex[20], invisible if: iq_uiCarrierIndex[20] = 0
    Rectangle (1,520 44x25), "20", invisible if: iq_uiCarrierIndex[20] = 0
END_VISUALIZATION

// LMC_PacDrive/Application/TemplateFullProgrammingFramework/Visualization/Multicarrier/Vis_ApplicationLogger
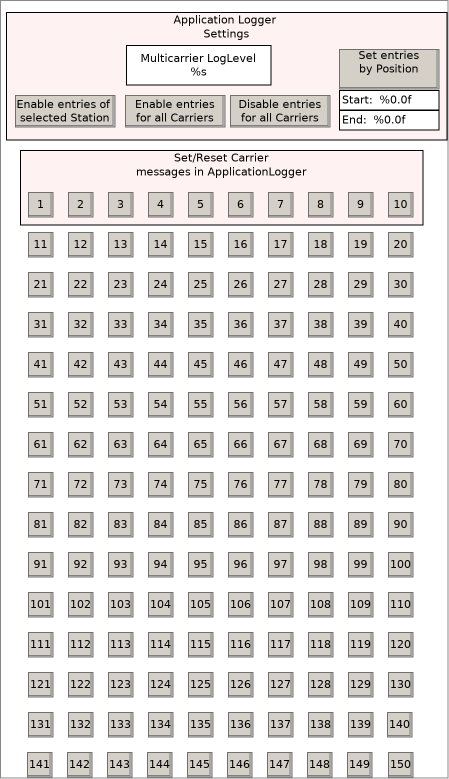
VISUALIZATION Vis_ApplicationLogger  // 449x779
    Rectangle (6,12 441x128), "Application Logger Settings", text variable: SR_MulticarrierModule.etLogLevelMcr
        OnMouseClick: write the text variable via Default
    Rectangle (126,45 145x40), "Multicarrier LogLevel %s", tooltip "0 - Nothing 50 - UserAction 70 - StatusMessage 80 - DebugMessage", text variable: SR_MulticarrierModule.etLogLevelMcr
        OnMouseClick: write the text variable via Default
    Rectangle (20,150 403x75), "Set/Reset Carrier messages in ApplicationLogger"
        p1126004900: SR_MultiCarriermodule.udiDeltaBottomY
    Button (15,95 100x32), "Enable entries of selected Station", colour toggle: GVL_Project.G_xEnableAplEntriesViaStation
        toggle GVL_Project.G_xEnableAplEntriesViaStation
    Button (125,95 100x32), "Enable entries for all Carriers", colour toggle: SR_MulticarrierModule.xSetForAllAplMsg
        toggle SR_MulticarrierModule.xSetForAllAplMsg
    Button (230,95 100x32), "Disable entries for all Carriers", colour toggle: SR_MulticarrierModule.xReSetForAllAplMsg
        toggle SR_MulticarrierModule.xReSetForAllAplMsg
    Button (28,192 25x25), "1", colour toggle: SR_MulticarrierModule.aifVisFeedback[1].ifFeedbackConfiguration.xApplicationLoggerEntriesActive, invisible if: SR_MulticarrierModule.ifMulticarrier.ifFeedback.ifFeedbackConfiguration.udiNumberOfCarriers < 1
        toggle SR_MulticarrierModule.xSetSingleAplMsg
        OnMouseDown: execute { SR_MulticarrierModule.udiSingleCarrierNr := 1; }
    Button (68,192 25x25), "2", colour toggle: SR_MulticarrierModule.aifVisFeedback[2].ifFeedbackConfiguration.xApplicationLoggerEntriesActive, invisible if: SR_MulticarrierModule.ifMulticarrier.ifFeedback.ifFeedbackConfiguration.udiNumberOfCarriers < 2
        toggle SR_MulticarrierModule.xSetSingleAplMsg
        OnMouseDown: execute { SR_MulticarrierModule.udiSingleCarrierNr := 2; }
    Button (108,192 25x25), "3", colour toggle: SR_MulticarrierModule.aifVisFeedback[3].ifFeedbackConfiguration.xApplicationLoggerEntriesActive, invisible if: SR_MulticarrierModule.ifMulticarrier.ifFeedback.ifFeedbackConfiguration.udiNumberOfCarriers < 3
        toggle SR_MulticarrierModule.xSetSingleAplMsg
        OnMouseDown: execute { SR_MulticarrierModule.udiSingleCarrierNr := 3; }
    Button (148,192 25x25), "4", colour toggle: SR_MulticarrierModule.aifVisFeedback[4].ifFeedbackConfiguration.xApplicationLoggerEntriesActive, invisible if: SR_MulticarrierModule.ifMulticarrier.ifFeedback.ifFeedbackConfiguration.udiNumberOfCarriers < 4
        toggle SR_MulticarrierModule.xSetSingleAplMsg
        OnMouseDown: execute { SR_MulticarrierModule.udiSingleCarrierNr := 4; }
    Button (188,192 25x25), "5", colour toggle: SR_MulticarrierModule.aifVisFeedback[5].ifFeedbackConfiguration.xApplicationLoggerEntriesActive, invisible if: SR_MulticarrierModule.ifMulticarrier.ifFeedback.ifFeedbackConfiguration.udiNumberOfCarriers < 5
        toggle SR_MulticarrierModule.xSetSingleAplMsg
        OnMouseDown: execute { SR_MulticarrierModule.udiSingleCarrierNr := 5; }
    Button (228,192 25x25), "6", colour toggle: SR_MulticarrierModule.aifVisFeedback[6].ifFeedbackConfiguration.xApplicationLoggerEntriesActive, invisible if: SR_MulticarrierModule.ifMulticarrier.ifFeedback.ifFeedbackConfiguration.udiNumberOfCarriers < 6
        toggle SR_MulticarrierModule.xSetSingleAplMsg
        OnMouseDown: execute { SR_MulticarrierModule.udiSingleCarrierNr := 6; }
    Button (268,192 25x25), "7", colour toggle: SR_MulticarrierModule.aifVisFeedback[7].ifFeedbackConfiguration.xApplicationLoggerEntriesActive, invisible if: SR_MulticarrierModule.ifMulticarrier.ifFeedback.ifFeedbackConfiguration.udiNumberOfCarriers < 7
        toggle SR_MulticarrierModule.xSetSingleAplMsg
        OnMouseDown: execute { SR_MulticarrierModule.udiSingleCarrierNr := 7; }
    Button (308,192 25x25), "8", colour toggle: SR_MulticarrierModule.aifVisFeedback[8].ifFeedbackConfiguration.xApplicationLoggerEntriesActive, invisible if: SR_MulticarrierModule.ifMulticarrier.ifFeedback.ifFeedbackConfiguration.udiNumberOfCarriers < 8
        toggle SR_MulticarrierModule.xSetSingleAplMsg
        OnMouseDown: execute { SR_MulticarrierModule.udiSingleCarrierNr := 8; }
    Button (348,192 25x25), "9", colour toggle: SR_MulticarrierModule.aifVisFeedback[9].ifFeedbackConfiguration.xApplicationLoggerEntriesActive, invisible if: SR_MulticarrierModule.ifMulticarrier.ifFeedback.ifFeedbackConfiguration.udiNumberOfCarriers < 9
        toggle SR_MulticarrierModule.xSetSingleAplMsg
        OnMouseDown: execute { SR_MulticarrierModule.udiSingleCarrierNr := 9; }
    Button (388,192 25x25), "10", colour toggle: SR_MulticarrierModule.aifVisFeedback[10].ifFeedbackConfiguration.xApplicationLoggerEntriesActive, invisible if: SR_MulticarrierModule.ifMulticarrier.ifFeedback.ifFeedbackConfiguration.udiNumberOfCarriers < 10
        toggle SR_MulticarrierModule.xSetSingleAplMsg
        OnMouseDown: execute { SR_MulticarrierModule.udiSingleCarrierNr := 10; }
    Button (28,232 25x25), "11", colour toggle: SR_MulticarrierModule.aifVisFeedback[11].ifFeedbackConfiguration.xApplicationLoggerEntriesActive, invisible if: SR_MulticarrierModule.ifMulticarrier.ifFeedback.ifFeedbackConfiguration.udiNumberOfCarriers < 11
        toggle SR_MulticarrierModule.xSetSingleAplMsg
        OnMouseDown: execute { SR_MulticarrierModule.udiSingleCarrierNr := 11; }
    Button (68,232 25x25), "12", colour toggle: SR_MulticarrierModule.aifVisFeedback[12].ifFeedbackConfiguration.xApplicationLoggerEntriesActive, invisible if: SR_MulticarrierModule.ifMulticarrier.ifFeedback.ifFeedbackConfiguration.udiNumberOfCarriers < 12
        toggle SR_MulticarrierModule.xSetSingleAplMsg
        OnMouseDown: execute { SR_MulticarrierModule.udiSingleCarrierNr := 12; }
    Button (108,232 25x25), "13", colour toggle: SR_MulticarrierModule.aifVisFeedback[13].ifFeedbackConfiguration.xApplicationLoggerEntriesActive, invisible if: SR_MulticarrierModule.ifMulticarrier.ifFeedback.ifFeedbackConfiguration.udiNumberOfCarriers < 13
        toggle SR_MulticarrierModule.xSetSingleAplMsg
        OnMouseDown: execute { SR_MulticarrierModule.udiSingleCarrierNr := 13; }
    Button (148,232 25x25), "14", colour toggle: SR_MulticarrierModule.aifVisFeedback[14].ifFeedbackConfiguration.xApplicationLoggerEntriesActive, invisible if: SR_MulticarrierModule.ifMulticarrier.ifFeedback.ifFeedbackConfiguration.udiNumberOfCarriers < 14
        toggle SR_MulticarrierModule.xSetSingleAplMsg
        OnMouseDown: execute { SR_MulticarrierModule.udiSingleCarrierNr := 14; }
    Button (188,232 25x25), "15", colour toggle: SR_MulticarrierModule.aifVisFeedback[15].ifFeedbackConfiguration.xApplicationLoggerEntriesActive, invisible if: SR_MulticarrierModule.ifMulticarrier.ifFeedback.ifFeedbackConfiguration.udiNumberOfCarriers < 15
        toggle SR_MulticarrierModule.xSetSingleAplMsg
        OnMouseDown: execute { SR_MulticarrierModule.udiSingleCarrierNr := 15; }
    Button (228,232 25x25), "16", colour toggle: SR_MulticarrierModule.aifVisFeedback[16].ifFeedbackConfiguration.xApplicationLoggerEntriesActive, invisible if: SR_MulticarrierModule.ifMulticarrier.ifFeedback.ifFeedbackConfiguration.udiNumberOfCarriers < 16
        toggle SR_MulticarrierModule.xSetSingleAplMsg
        OnMouseDown: execute { SR_MulticarrierModule.udiSingleCarrierNr := 16; }
    Button (268,232 25x25), "17", colour toggle: SR_MulticarrierModule.aifVisFeedback[17].ifFeedbackConfiguration.xApplicationLoggerEntriesActive, invisible if: SR_MulticarrierModule.ifMulticarrier.ifFeedback.ifFeedbackConfiguration.udiNumberOfCarriers < 17
        toggle SR_MulticarrierModule.xSetSingleAplMsg
        OnMouseDown: execute { SR_MulticarrierModule.udiSingleCarrierNr := 17; }
    Button (308,232 25x25), "18", colour toggle: SR_MulticarrierModule.aifVisFeedback[18].ifFeedbackConfiguration.xApplicationLoggerEntriesActive, invisible if: SR_MulticarrierModule.ifMulticarrier.ifFeedback.ifFeedbackConfiguration.udiNumberOfCarriers < 18
        toggle SR_MulticarrierModule.xSetSingleAplMsg
        OnMouseDown: execute { SR_MulticarrierModule.udiSingleCarrierNr := 18; }
    Button (348,232 25x25), "19", colour toggle: SR_MulticarrierModule.aifVisFeedback[19].ifFeedbackConfiguration.xApplicationLoggerEntriesActive, invisible if: SR_MulticarrierModule.ifMulticarrier.ifFeedback.ifFeedbackConfiguration.udiNumberOfCarriers < 19
        toggle SR_MulticarrierModule.xSetSingleAplMsg
        OnMouseDown: execute { SR_MulticarrierModule.udiSingleCarrierNr := 19; }
    Button (388,232 25x25), "20", colour toggle: SR_MulticarrierModule.aifVisFeedback[20].ifFeedbackConfiguration.xApplicationLoggerEntriesActive, invisible if: SR_MulticarrierModule.ifMulticarrier.ifFeedback.ifFeedbackConfiguration.udiNumberOfCarriers < 20
        toggle SR_MulticarrierModule.xSetSingleAplMsg
        OnMouseDown: execute { SR_MulticarrierModule.udiSingleCarrierNr := 20; }
    Button (28,272 25x25), "21", colour toggle: SR_MulticarrierModule.aifVisFeedback[21].ifFeedbackConfiguration.xApplicationLoggerEntriesActive, invisible if: SR_MulticarrierModule.ifMulticarrier.ifFeedback.ifFeedbackConfiguration.udiNumberOfCarriers < 21
        toggle SR_MulticarrierModule.xSetSingleAplMsg
        OnMouseDown: execute { SR_MulticarrierModule.udiSingleCarrierNr := 21; }
    Button (68,272 25x25), "22", colour toggle: SR_MulticarrierModule.aifVisFeedback[22].ifFeedbackConfiguration.xApplicationLoggerEntriesActive, invisible if: SR_MulticarrierModule.ifMulticarrier.ifFeedback.ifFeedbackConfiguration.udiNumberOfCarriers < 22
        toggle SR_MulticarrierModule.xSetSingleAplMsg
        OnMouseDown: execute { SR_MulticarrierModule.udiSingleCarrierNr := 22; }
    Button (108,272 25x25), "23", colour toggle: SR_MulticarrierModule.aifVisFeedback[23].ifFeedbackConfiguration.xApplicationLoggerEntriesActive, invisible if: SR_MulticarrierModule.ifMulticarrier.ifFeedback.ifFeedbackConfiguration.udiNumberOfCarriers < 23
        toggle SR_MulticarrierModule.xSetSingleAplMsg
        OnMouseDown: execute { SR_MulticarrierModule.udiSingleCarrierNr := 23; }
    Button (148,272 25x25), "24", colour toggle: SR_MulticarrierModule.aifVisFeedback[24].ifFeedbackConfiguration.xApplicationLoggerEntriesActive, invisible if: SR_MulticarrierModule.ifMulticarrier.ifFeedback.ifFeedbackConfiguration.udiNumberOfCarriers < 24
        toggle SR_MulticarrierModule.xSetSingleAplMsg
        OnMouseDown: execute { SR_MulticarrierModule.udiSingleCarrierNr := 24; }
    Button (188,272 25x25), "25", colour toggle: SR_MulticarrierModule.aifVisFeedback[25].ifFeedbackConfiguration.xApplicationLoggerEntriesActive, invisible if: SR_MulticarrierModule.ifMulticarrier.ifFeedback.ifFeedbackConfiguration.udiNumberOfCarriers < 25
        toggle SR_MulticarrierModule.xSetSingleAplMsg
        OnMouseDown: execute { SR_MulticarrierModule.udiSingleCarrierNr := 25; }
    Button (228,272 25x25), "26", colour toggle: SR_MulticarrierModule.aifVisFeedback[26].ifFeedbackConfiguration.xApplicationLoggerEntriesActive, invisible if: SR_MulticarrierModule.ifMulticarrier.ifFeedback.ifFeedbackConfiguration.udiNumberOfCarriers < 26
        toggle SR_MulticarrierModule.xSetSingleAplMsg
        OnMouseDown: execute { SR_MulticarrierModule.udiSingleCarrierNr := 26; }
    Button (268,272 25x25), "27", colour toggle: SR_MulticarrierModule.aifVisFeedback[27].ifFeedbackConfiguration.xApplicationLoggerEntriesActive, invisible if: SR_MulticarrierModule.ifMulticarrier.ifFeedback.ifFeedbackConfiguration.udiNumberOfCarriers < 27
        toggle SR_MulticarrierModule.xSetSingleAplMsg
        OnMouseDown: execute { SR_MulticarrierModule.udiSingleCarrierNr := 27; }
    Button (308,272 25x25), "28", colour toggle: SR_MulticarrierModule.aifVisFeedback[28].ifFeedbackConfiguration.xApplicationLoggerEntriesActive, invisible if: SR_MulticarrierModule.ifMulticarrier.ifFeedback.ifFeedbackConfiguration.udiNumberOfCarriers < 28
        toggle SR_MulticarrierModule.xSetSingleAplMsg
        OnMouseDown: execute { SR_MulticarrierModule.udiSingleCarrierNr := 28; }
    Button (348,272 25x25), "29", colour toggle: SR_MulticarrierModule.aifVisFeedback[29].ifFeedbackConfiguration.xApplicationLoggerEntriesActive, invisible if: SR_MulticarrierModule.ifMulticarrier.ifFeedback.ifFeedbackConfiguration.udiNumberOfCarriers < 29
        toggle SR_MulticarrierModule.xSetSingleAplMsg
        OnMouseDown: execute { SR_MulticarrierModule.udiSingleCarrierNr := 29; }
    Button (388,272 25x25), "30", colour toggle: SR_MulticarrierModule.aifVisFeedback[30].ifFeedbackConfiguration.xApplicationLoggerEntriesActive, invisible if: SR_MulticarrierModule.ifMulticarrier.ifFeedback.ifFeedbackConfiguration.udiNumberOfCarriers < 30
        toggle SR_MulticarrierModule.xSetSingleAplMsg
        OnMouseDown: execute { SR_MulticarrierModule.udiSingleCarrierNr := 30; }
    Button (28,312 25x25), "31", colour toggle: SR_MulticarrierModule.aifVisFeedback[31].ifFeedbackConfiguration.xApplicationLoggerEntriesActive, invisible if: SR_MulticarrierModule.ifMulticarrier.ifFeedback.ifFeedbackConfiguration.udiNumberOfCarriers < 31
        toggle SR_MulticarrierModule.xSetSingleAplMsg
        OnMouseDown: execute { SR_MulticarrierModule.udiSingleCarrierNr := 31; }
    Button (68,312 25x25), "32", colour toggle: SR_MulticarrierModule.aifVisFeedback[32].ifFeedbackConfiguration.xApplicationLoggerEntriesActive, invisible if: SR_MulticarrierModule.ifMulticarrier.ifFeedback.ifFeedbackConfiguration.udiNumberOfCarriers < 32
        toggle SR_MulticarrierModule.xSetSingleAplMsg
        OnMouseDown: execute { SR_MulticarrierModule.udiSingleCarrierNr := 32; }
    Button (108,312 25x25), "33", colour toggle: SR_MulticarrierModule.aifVisFeedback[33].ifFeedbackConfiguration.xApplicationLoggerEntriesActive, invisible if: SR_MulticarrierModule.ifMulticarrier.ifFeedback.ifFeedbackConfiguration.udiNumberOfCarriers < 33
        toggle SR_MulticarrierModule.xSetSingleAplMsg
        OnMouseDown: execute { SR_MulticarrierModule.udiSingleCarrierNr := 33; }
    Button (148,312 25x25), "34", colour toggle: SR_MulticarrierModule.aifVisFeedback[34].ifFeedbackConfiguration.xApplicationLoggerEntriesActive, invisible if: SR_MulticarrierModule.ifMulticarrier.ifFeedback.ifFeedbackConfiguration.udiNumberOfCarriers < 34
        toggle SR_MulticarrierModule.xSetSingleAplMsg
        OnMouseDown: execute { SR_MulticarrierModule.udiSingleCarrierNr := 34; }
    Button (188,312 25x25), "35", colour toggle: SR_MulticarrierModule.aifVisFeedback[35].ifFeedbackConfiguration.xApplicationLoggerEntriesActive, invisible if: SR_MulticarrierModule.ifMulticarrier.ifFeedback.ifFeedbackConfiguration.udiNumberOfCarriers < 35
        toggle SR_MulticarrierModule.xSetSingleAplMsg
        OnMouseDown: execute { SR_MulticarrierModule.udiSingleCarrierNr := 35; }
    Button (228,312 25x25), "36", colour toggle: SR_MulticarrierModule.aifVisFeedback[36].ifFeedbackConfiguration.xApplicationLoggerEntriesActive, invisible if: SR_MulticarrierModule.ifMulticarrier.ifFeedback.ifFeedbackConfiguration.udiNumberOfCarriers < 36
        toggle SR_MulticarrierModule.xSetSingleAplMsg
        OnMouseDown: execute { SR_MulticarrierModule.udiSingleCarrierNr := 36; }
    Button (268,312 25x25), "37", colour toggle: SR_MulticarrierModule.aifVisFeedback[37].ifFeedbackConfiguration.xApplicationLoggerEntriesActive, invisible if: SR_MulticarrierModule.ifMulticarrier.ifFeedback.ifFeedbackConfiguration.udiNumberOfCarriers < 37
        toggle SR_MulticarrierModule.xSetSingleAplMsg
        OnMouseDown: execute { SR_MulticarrierModule.udiSingleCarrierNr := 37; }
    Button (308,312 25x25), "38", colour toggle: SR_MulticarrierModule.aifVisFeedback[38].ifFeedbackConfiguration.xApplicationLoggerEntriesActive, invisible if: SR_MulticarrierModule.ifMulticarrier.ifFeedback.ifFeedbackConfiguration.udiNumberOfCarriers < 38
        toggle SR_MulticarrierModule.xSetSingleAplMsg
        OnMouseDown: execute { SR_MulticarrierModule.udiSingleCarrierNr := 38; }
    Button (348,312 25x25), "39", colour toggle: SR_MulticarrierModule.aifVisFeedback[39].ifFeedbackConfiguration.xApplicationLoggerEntriesActive, invisible if: SR_MulticarrierModule.ifMulticarrier.ifFeedback.ifFeedbackConfiguration.udiNumberOfCarriers < 39
        toggle SR_MulticarrierModule.xSetSingleAplMsg
        OnMouseDown: execute { SR_MulticarrierModule.udiSingleCarrierNr := 39; }
    Button (388,312 25x25), "40", colour toggle: SR_MulticarrierModule.aifVisFeedback[40].ifFeedbackConfiguration.xApplicationLoggerEntriesActive, invisible if: SR_MulticarrierModule.ifMulticarrier.ifFeedback.ifFeedbackConfiguration.udiNumberOfCarriers < 40
        toggle SR_MulticarrierModule.xSetSingleAplMsg
        OnMouseDown: execute { SR_MulticarrierModule.udiSingleCarrierNr := 40; }
    Button (28,352 25x25), "41", colour toggle: SR_MulticarrierModule.aifVisFeedback[41].ifFeedbackConfiguration.xApplicationLoggerEntriesActive, invisible if: SR_MulticarrierModule.ifMulticarrier.ifFeedback.ifFeedbackConfiguration.udiNumberOfCarriers < 41
        toggle SR_MulticarrierModule.xSetSingleAplMsg
        OnMouseDown: execute { SR_MulticarrierModule.udiSingleCarrierNr := 41; }
    Button (68,352 25x25), "42", colour toggle: SR_MulticarrierModule.aifVisFeedback[42].ifFeedbackConfiguration.xApplicationLoggerEntriesActive, invisible if: SR_MulticarrierModule.ifMulticarrier.ifFeedback.ifFeedbackConfiguration.udiNumberOfCarriers < 42
        toggle SR_MulticarrierModule.xSetSingleAplMsg
        OnMouseDown: execute { SR_MulticarrierModule.udiSingleCarrierNr := 42; }
    Button (108,352 25x25), "43", colour toggle: SR_MulticarrierModule.aifVisFeedback[43].ifFeedbackConfiguration.xApplicationLoggerEntriesActive, invisible if: SR_MulticarrierModule.ifMulticarrier.ifFeedback.ifFeedbackConfiguration.udiNumberOfCarriers < 43
        toggle SR_MulticarrierModule.xSetSingleAplMsg
        OnMouseDown: execute { SR_MulticarrierModule.udiSingleCarrierNr := 43; }
    Button (148,352 25x25), "44", colour toggle: SR_MulticarrierModule.aifVisFeedback[44].ifFeedbackConfiguration.xApplicationLoggerEntriesActive, invisible if: SR_MulticarrierModule.ifMulticarrier.ifFeedback.ifFeedbackConfiguration.udiNumberOfCarriers < 44
        toggle SR_MulticarrierModule.xSetSingleAplMsg
        OnMouseDown: execute { SR_MulticarrierModule.udiSingleCarrierNr := 44; }
    Button (188,352 25x25), "45", colour toggle: SR_MulticarrierModule.aifVisFeedback[45].ifFeedbackConfiguration.xApplicationLoggerEntriesActive, invisible if: SR_MulticarrierModule.ifMulticarrier.ifFeedback.ifFeedbackConfiguration.udiNumberOfCarriers < 45
        toggle SR_MulticarrierModule.xSetSingleAplMsg
        OnMouseDown: execute { SR_MulticarrierModule.udiSingleCarrierNr := 45; }
    Button (228,352 25x25), "46", colour toggle: SR_MulticarrierModule.aifVisFeedback[46].ifFeedbackConfiguration.xApplicationLoggerEntriesActive, invisible if: SR_MulticarrierModule.ifMulticarrier.ifFeedback.ifFeedbackConfiguration.udiNumberOfCarriers < 46
        toggle SR_MulticarrierModule.xSetSingleAplMsg
        OnMouseDown: execute { SR_MulticarrierModule.udiSingleCarrierNr := 46; }
    Button (268,352 25x25), "47", colour toggle: SR_MulticarrierModule.aifVisFeedback[47].ifFeedbackConfiguration.xApplicationLoggerEntriesActive, invisible if: SR_MulticarrierModule.ifMulticarrier.ifFeedback.ifFeedbackConfiguration.udiNumberOfCarriers < 47
        toggle SR_MulticarrierModule.xSetSingleAplMsg
        OnMouseDown: execute { SR_MulticarrierModule.udiSingleCarrierNr := 47; }
    Button (308,352 25x25), "48", colour toggle: SR_MulticarrierModule.aifVisFeedback[48].ifFeedbackConfiguration.xApplicationLoggerEntriesActive, invisible if: SR_MulticarrierModule.ifMulticarrier.ifFeedback.ifFeedbackConfiguration.udiNumberOfCarriers < 48
        toggle SR_MulticarrierModule.xSetSingleAplMsg
        OnMouseDown: execute { SR_MulticarrierModule.udiSingleCarrierNr := 48; }
    Button (348,352 25x25), "49", colour toggle: SR_MulticarrierModule.aifVisFeedback[49].ifFeedbackConfiguration.xApplicationLoggerEntriesActive, invisible if: SR_MulticarrierModule.ifMulticarrier.ifFeedback.ifFeedbackConfiguration.udiNumberOfCarriers < 49
        toggle SR_MulticarrierModule.xSetSingleAplMsg
        OnMouseDown: execute { SR_MulticarrierModule.udiSingleCarrierNr := 49; }
    Button (388,352 25x25), "50", colour toggle: SR_MulticarrierModule.aifVisFeedback[50].ifFeedbackConfiguration.xApplicationLoggerEntriesActive, invisible if: SR_MulticarrierModule.ifMulticarrier.ifFeedback.ifFeedbackConfiguration.udiNumberOfCarriers < 50
        toggle SR_MulticarrierModule.xSetSingleAplMsg
        OnMouseDown: execute { SR_MulticarrierModule.udiSingleCarrierNr := 50; }
    Button (28,392 25x25), "51", colour toggle: SR_MulticarrierModule.aifVisFeedback[51].ifFeedbackConfiguration.xApplicationLoggerEntriesActive, invisible if: SR_MulticarrierModule.ifMulticarrier.ifFeedback.ifFeedbackConfiguration.udiNumberOfCarriers < 51
        toggle SR_MulticarrierModule.xSetSingleAplMsg
        OnMouseDown: execute { SR_MulticarrierModule.udiSingleCarrierNr := 51; }
    Button (68,392 25x25), "52", colour toggle: SR_MulticarrierModule.aifVisFeedback[52].ifFeedbackConfiguration.xApplicationLoggerEntriesActive, invisible if: SR_MulticarrierModule.ifMulticarrier.ifFeedback.ifFeedbackConfiguration.udiNumberOfCarriers < 52
        toggle SR_MulticarrierModule.xSetSingleAplMsg
        OnMouseDown: execute { SR_MulticarrierModule.udiSingleCarrierNr := 52; }
    Button (108,392 25x25), "53", colour toggle: SR_MulticarrierModule.aifVisFeedback[53].ifFeedbackConfiguration.xApplicationLoggerEntriesActive, invisible if: SR_MulticarrierModule.ifMulticarrier.ifFeedback.ifFeedbackConfiguration.udiNumberOfCarriers < 53
        toggle SR_MulticarrierModule.xSetSingleAplMsg
        OnMouseDown: execute { SR_MulticarrierModule.udiSingleCarrierNr := 53; }
    Button (148,392 25x25), "54", colour toggle: SR_MulticarrierModule.aifVisFeedback[54].ifFeedbackConfiguration.xApplicationLoggerEntriesActive, invisible if: SR_MulticarrierModule.ifMulticarrier.ifFeedback.ifFeedbackConfiguration.udiNumberOfCarriers < 54
        toggle SR_MulticarrierModule.xSetSingleAplMsg
        OnMouseDown: execute { SR_MulticarrierModule.udiSingleCarrierNr := 54; }
    Button (188,392 25x25), "55", colour toggle: SR_MulticarrierModule.aifVisFeedback[55].ifFeedbackConfiguration.xApplicationLoggerEntriesActive, invisible if: SR_MulticarrierModule.ifMulticarrier.ifFeedback.ifFeedbackConfiguration.udiNumberOfCarriers < 55
        toggle SR_MulticarrierModule.xSetSingleAplMsg
        OnMouseDown: execute { SR_MulticarrierModule.udiSingleCarrierNr := 55; }
    Button (228,392 25x25), "56", colour toggle: SR_MulticarrierModule.aifVisFeedback[56].ifFeedbackConfiguration.xApplicationLoggerEntriesActive, invisible if: SR_MulticarrierModule.ifMulticarrier.ifFeedback.ifFeedbackConfiguration.udiNumberOfCarriers < 56
        toggle SR_MulticarrierModule.xSetSingleAplMsg
        OnMouseDown: execute { SR_MulticarrierModule.udiSingleCarrierNr := 56; }
    Button (268,392 25x25), "57", colour toggle: SR_MulticarrierModule.aifVisFeedback[57].ifFeedbackConfiguration.xApplicationLoggerEntriesActive, invisible if: SR_MulticarrierModule.ifMulticarrier.ifFeedback.ifFeedbackConfiguration.udiNumberOfCarriers < 57
        toggle SR_MulticarrierModule.xSetSingleAplMsg
        OnMouseDown: execute { SR_MulticarrierModule.udiSingleCarrierNr := 57; }
    Button (308,392 25x25), "58", colour toggle: SR_MulticarrierModule.aifVisFeedback[58].ifFeedbackConfiguration.xApplicationLoggerEntriesActive, invisible if: SR_MulticarrierModule.ifMulticarrier.ifFeedback.ifFeedbackConfiguration.udiNumberOfCarriers < 58
        toggle SR_MulticarrierModule.xSetSingleAplMsg
        OnMouseDown: execute { SR_MulticarrierModule.udiSingleCarrierNr := 58; }
    Button (348,392 25x25), "59", colour toggle: SR_MulticarrierModule.aifVisFeedback[59].ifFeedbackConfiguration.xApplicationLoggerEntriesActive, invisible if: SR_MulticarrierModule.ifMulticarrier.ifFeedback.ifFeedbackConfiguration.udiNumberOfCarriers < 59
        toggle SR_MulticarrierModule.xSetSingleAplMsg
        OnMouseDown: execute { SR_MulticarrierModule.udiSingleCarrierNr := 59; }
    Button (388,392 25x25), "60", colour toggle: SR_MulticarrierModule.aifVisFeedback[60].ifFeedbackConfiguration.xApplicationLoggerEntriesActive, invisible if: SR_MulticarrierModule.ifMulticarrier.ifFeedback.ifFeedbackConfiguration.udiNumberOfCarriers < 60
        toggle SR_MulticarrierModule.xSetSingleAplMsg
        OnMouseDown: execute { SR_MulticarrierModule.udiSingleCarrierNr := 60; }
    Button (28,432 25x25), "61", colour toggle: SR_MulticarrierModule.aifVisFeedback[61].ifFeedbackConfiguration.xApplicationLoggerEntriesActive, invisible if: SR_MulticarrierModule.ifMulticarrier.ifFeedback.ifFeedbackConfiguration.udiNumberOfCarriers < 61
        toggle SR_MulticarrierModule.xSetSingleAplMsg
        OnMouseDown: execute { SR_MulticarrierModule.udiSingleCarrierNr := 61; }
    Button (68,432 25x25), "62", colour toggle: SR_MulticarrierModule.aifVisFeedback[62].ifFeedbackConfiguration.xApplicationLoggerEntriesActive, invisible if: SR_MulticarrierModule.ifMulticarrier.ifFeedback.ifFeedbackConfiguration.udiNumberOfCarriers < 62
        toggle SR_MulticarrierModule.xSetSingleAplMsg
        OnMouseDown: execute { SR_MulticarrierModule.udiSingleCarrierNr := 62; }
    Button (108,432 25x25), "63", colour toggle: SR_MulticarrierModule.aifVisFeedback[63].ifFeedbackConfiguration.xApplicationLoggerEntriesActive, invisible if: SR_MulticarrierModule.ifMulticarrier.ifFeedback.ifFeedbackConfiguration.udiNumberOfCarriers < 63
        toggle SR_MulticarrierModule.xSetSingleAplMsg
        OnMouseDown: execute { SR_MulticarrierModule.udiSingleCarrierNr := 63; }
    Button (148,432 25x25), "64", colour toggle: SR_MulticarrierModule.aifVisFeedback[64].ifFeedbackConfiguration.xApplicationLoggerEntriesActive, invisible if: SR_MulticarrierModule.ifMulticarrier.ifFeedback.ifFeedbackConfiguration.udiNumberOfCarriers < 64
        toggle SR_MulticarrierModule.xSetSingleAplMsg
        OnMouseDown: execute { SR_MulticarrierModule.udiSingleCarrierNr := 64; }
    Button (188,432 25x25), "65", colour toggle: SR_MulticarrierModule.aifVisFeedback[65].ifFeedbackConfiguration.xApplicationLoggerEntriesActive, invisible if: SR_MulticarrierModule.ifMulticarrier.ifFeedback.ifFeedbackConfiguration.udiNumberOfCarriers < 65
        toggle SR_MulticarrierModule.xSetSingleAplMsg
        OnMouseDown: execute { SR_MulticarrierModule.udiSingleCarrierNr := 65; }
    Button (228,432 25x25), "66", colour toggle: SR_MulticarrierModule.aifVisFeedback[66].ifFeedbackConfiguration.xApplicationLoggerEntriesActive, invisible if: SR_MulticarrierModule.ifMulticarrier.ifFeedback.ifFeedbackConfiguration.udiNumberOfCarriers < 66
        toggle SR_MulticarrierModule.xSetSingleAplMsg
        OnMouseDown: execute { SR_MulticarrierModule.udiSingleCarrierNr := 66; }
    Button (268,432 25x25), "67", colour toggle: SR_MulticarrierModule.aifVisFeedback[67].ifFeedbackConfiguration.xApplicationLoggerEntriesActive, invisible if: SR_MulticarrierModule.ifMulticarrier.ifFeedback.ifFeedbackConfiguration.udiNumberOfCarriers < 67
        toggle SR_MulticarrierModule.xSetSingleAplMsg
        OnMouseDown: execute { SR_MulticarrierModule.udiSingleCarrierNr := 67; }
    Button (308,432 25x25), "68", colour toggle: SR_MulticarrierModule.aifVisFeedback[68].ifFeedbackConfiguration.xApplicationLoggerEntriesActive, invisible if: SR_MulticarrierModule.ifMulticarrier.ifFeedback.ifFeedbackConfiguration.udiNumberOfCarriers < 68
        toggle SR_MulticarrierModule.xSetSingleAplMsg
        OnMouseDown: execute { SR_MulticarrierModule.udiSingleCarrierNr := 68; }
    Button (348,432 25x25), "69", colour toggle: SR_MulticarrierModule.aifVisFeedback[69].ifFeedbackConfiguration.xApplicationLoggerEntriesActive, invisible if: SR_MulticarrierModule.ifMulticarrier.ifFeedback.ifFeedbackConfiguration.udiNumberOfCarriers < 69
        toggle SR_MulticarrierModule.xSetSingleAplMsg
        OnMouseDown: execute { SR_MulticarrierModule.udiSingleCarrierNr := 69; }
    Button (388,432 25x25), "70", colour toggle: SR_MulticarrierModule.aifVisFeedback[70].ifFeedbackConfiguration.xApplicationLoggerEntriesActive, invisible if: SR_MulticarrierModule.ifMulticarrier.ifFeedback.ifFeedbackConfiguration.udiNumberOfCarriers < 70
        toggle SR_MulticarrierModule.xSetSingleAplMsg
        OnMouseDown: execute { SR_MulticarrierModule.udiSingleCarrierNr := 70; }
    Button (28,472 25x25), "71", colour toggle: SR_MulticarrierModule.aifVisFeedback[71].ifFeedbackConfiguration.xApplicationLoggerEntriesActive, invisible if: SR_MulticarrierModule.ifMulticarrier.ifFeedback.ifFeedbackConfiguration.udiNumberOfCarriers < 71
        toggle SR_MulticarrierModule.xSetSingleAplMsg
        OnMouseDown: execute { SR_MulticarrierModule.udiSingleCarrierNr := 71; }
    Button (68,472 25x25), "72", colour toggle: SR_MulticarrierModule.aifVisFeedback[72].ifFeedbackConfiguration.xApplicationLoggerEntriesActive, invisible if: SR_MulticarrierModule.ifMulticarrier.ifFeedback.ifFeedbackConfiguration.udiNumberOfCarriers < 72
        toggle SR_MulticarrierModule.xSetSingleAplMsg
        OnMouseDown: execute { SR_MulticarrierModule.udiSingleCarrierNr := 72; }
    Button (108,472 25x25), "73", colour toggle: SR_MulticarrierModule.aifVisFeedback[73].ifFeedbackConfiguration.xApplicationLoggerEntriesActive, invisible if: SR_MulticarrierModule.ifMulticarrier.ifFeedback.ifFeedbackConfiguration.udiNumberOfCarriers < 73
        toggle SR_MulticarrierModule.xSetSingleAplMsg
        OnMouseDown: execute { SR_MulticarrierModule.udiSingleCarrierNr := 73; }
    Button (148,472 25x25), "74", colour toggle: SR_MulticarrierModule.aifVisFeedback[74].ifFeedbackConfiguration.xApplicationLoggerEntriesActive, invisible if: SR_MulticarrierModule.ifMulticarrier.ifFeedback.ifFeedbackConfiguration.udiNumberOfCarriers < 74
        toggle SR_MulticarrierModule.xSetSingleAplMsg
        OnMouseDown: execute { SR_MulticarrierModule.udiSingleCarrierNr := 74; }
    Button (188,472 25x25), "75", colour toggle: SR_MulticarrierModule.aifVisFeedback[75].ifFeedbackConfiguration.xApplicationLoggerEntriesActive, invisible if: SR_MulticarrierModule.ifMulticarrier.ifFeedback.ifFeedbackConfiguration.udiNumberOfCarriers < 75
        toggle SR_MulticarrierModule.xSetSingleAplMsg
        OnMouseDown: execute { SR_MulticarrierModule.udiSingleCarrierNr := 75; }
    Button (228,472 25x25), "76", colour toggle: SR_MulticarrierModule.aifVisFeedback[76].ifFeedbackConfiguration.xApplicationLoggerEntriesActive, invisible if: SR_MulticarrierModule.ifMulticarrier.ifFeedback.ifFeedbackConfiguration.udiNumberOfCarriers < 77
        toggle SR_MulticarrierModule.xSetSingleAplMsg
        OnMouseDown: execute { SR_MulticarrierModule.udiSingleCarrierNr := 76; }
    Button (268,472 25x25), "77", colour toggle: SR_MulticarrierModule.aifVisFeedback[77].ifFeedbackConfiguration.xApplicationLoggerEntriesActive, invisible if: SR_MulticarrierModule.ifMulticarrier.ifFeedback.ifFeedbackConfiguration.udiNumberOfCarriers < 77
        toggle SR_MulticarrierModule.xSetSingleAplMsg
        OnMouseDown: execute { SR_MulticarrierModule.udiSingleCarrierNr := 77; }
    Button (308,472 25x25), "78", colour toggle: SR_MulticarrierModule.aifVisFeedback[78].ifFeedbackConfiguration.xApplicationLoggerEntriesActive, invisible if: SR_MulticarrierModule.ifMulticarrier.ifFeedback.ifFeedbackConfiguration.udiNumberOfCarriers < 78
        toggle SR_MulticarrierModule.xSetSingleAplMsg
        OnMouseDown: execute { SR_MulticarrierModule.udiSingleCarrierNr := 78; }
    Button (348,472 25x25), "79", colour toggle: SR_MulticarrierModule.aifVisFeedback[79].ifFeedbackConfiguration.xApplicationLoggerEntriesActive, invisible if: SR_MulticarrierModule.ifMulticarrier.ifFeedback.ifFeedbackConfiguration.udiNumberOfCarriers < 79
        toggle SR_MulticarrierModule.xSetSingleAplMsg
        OnMouseDown: execute { SR_MulticarrierModule.udiSingleCarrierNr := 79; }
    Button (388,472 25x25), "80", colour toggle: SR_MulticarrierModule.aifVisFeedback[80].ifFeedbackConfiguration.xApplicationLoggerEntriesActive, invisible if: SR_MulticarrierModule.ifMulticarrier.ifFeedback.ifFeedbackConfiguration.udiNumberOfCarriers < 80
        toggle SR_MulticarrierModule.xSetSingleAplMsg
        OnMouseDown: execute { SR_MulticarrierModule.udiSingleCarrierNr := 80; }
    Button (28,512 25x25), "81", colour toggle: SR_MulticarrierModule.aifVisFeedback[81].ifFeedbackConfiguration.xApplicationLoggerEntriesActive, invisible if: SR_MulticarrierModule.ifMulticarrier.ifFeedback.ifFeedbackConfiguration.udiNumberOfCarriers < 81
        toggle SR_MulticarrierModule.xSetSingleAplMsg
        OnMouseDown: execute { SR_MulticarrierModule.udiSingleCarrierNr := 81; }
    Button (68,512 25x25), "82", colour toggle: SR_MulticarrierModule.aifVisFeedback[82].ifFeedbackConfiguration.xApplicationLoggerEntriesActive, invisible if: SR_MulticarrierModule.ifMulticarrier.ifFeedback.ifFeedbackConfiguration.udiNumberOfCarriers < 82
        toggle SR_MulticarrierModule.xSetSingleAplMsg
        OnMouseDown: execute { SR_MulticarrierModule.udiSingleCarrierNr := 82; }
    Button (108,512 25x25), "83", colour toggle: SR_MulticarrierModule.aifVisFeedback[83].ifFeedbackConfiguration.xApplicationLoggerEntriesActive, invisible if: SR_MulticarrierModule.ifMulticarrier.ifFeedback.ifFeedbackConfiguration.udiNumberOfCarriers < 83
        toggle SR_MulticarrierModule.xSetSingleAplMsg
        OnMouseDown: execute { SR_MulticarrierModule.udiSingleCarrierNr := 83; }
    Button (148,512 25x25), "84", colour toggle: SR_MulticarrierModule.aifVisFeedback[84].ifFeedbackConfiguration.xApplicationLoggerEntriesActive, invisible if: SR_MulticarrierModule.ifMulticarrier.ifFeedback.ifFeedbackConfiguration.udiNumberOfCarriers < 84
        toggle SR_MulticarrierModule.xSetSingleAplMsg
        OnMouseDown: execute { SR_MulticarrierModule.udiSingleCarrierNr := 84; }
    Button (188,512 25x25), "85", colour toggle: SR_MulticarrierModule.aifVisFeedback[85].ifFeedbackConfiguration.xApplicationLoggerEntriesActive, invisible if: SR_MulticarrierModule.ifMulticarrier.ifFeedback.ifFeedbackConfiguration.udiNumberOfCarriers < 85
        toggle SR_MulticarrierModule.xSetSingleAplMsg
        OnMouseDown: execute { SR_MulticarrierModule.udiSingleCarrierNr := 85; }
    Button (228,512 25x25), "86", colour toggle: SR_MulticarrierModule.aifVisFeedback[86].ifFeedbackConfiguration.xApplicationLoggerEntriesActive, invisible if: SR_MulticarrierModule.ifMulticarrier.ifFeedback.ifFeedbackConfiguration.udiNumberOfCarriers < 88
        toggle SR_MulticarrierModule.xSetSingleAplMsg
        OnMouseDown: execute { SR_MulticarrierModule.udiSingleCarrierNr := 86; }
    Button (268,512 25x25), "87", colour toggle: SR_MulticarrierModule.aifVisFeedback[87].ifFeedbackConfiguration.xApplicationLoggerEntriesActive, invisible if: SR_MulticarrierModule.ifMulticarrier.ifFeedback.ifFeedbackConfiguration.udiNumberOfCarriers < 88
        toggle SR_MulticarrierModule.xSetSingleAplMsg
        OnMouseDown: execute { SR_MulticarrierModule.udiSingleCarrierNr := 87; }
    Button (308,512 25x25), "88", colour toggle: SR_MulticarrierModule.aifVisFeedback[88].ifFeedbackConfiguration.xApplicationLoggerEntriesActive, invisible if: SR_MulticarrierModule.ifMulticarrier.ifFeedback.ifFeedbackConfiguration.udiNumberOfCarriers < 88
        toggle SR_MulticarrierModule.xSetSingleAplMsg
        OnMouseDown: execute { SR_MulticarrierModule.udiSingleCarrierNr := 88; }
    Button (348,512 25x25), "89", colour toggle: SR_MulticarrierModule.aifVisFeedback[89].ifFeedbackConfiguration.xApplicationLoggerEntriesActive, invisible if: SR_MulticarrierModule.ifMulticarrier.ifFeedback.ifFeedbackConfiguration.udiNumberOfCarriers < 89
        toggle SR_MulticarrierModule.xSetSingleAplMsg
        OnMouseDown: execute { SR_MulticarrierModule.udiSingleCarrierNr := 89; }
    Button (388,512 25x25), "90", colour toggle: SR_MulticarrierModule.aifVisFeedback[90].ifFeedbackConfiguration.xApplicationLoggerEntriesActive, invisible if: SR_MulticarrierModule.ifMulticarrier.ifFeedback.ifFeedbackConfiguration.udiNumberOfCarriers < 90
        toggle SR_MulticarrierModule.xSetSingleAplMsg
        OnMouseDown: execute { SR_MulticarrierModule.udiSingleCarrierNr := 90; }
    Button (28,552 25x25), "91", colour toggle: SR_MulticarrierModule.aifVisFeedback[91].ifFeedbackConfiguration.xApplicationLoggerEntriesActive, invisible if: SR_MulticarrierModule.ifMulticarrier.ifFeedback.ifFeedbackConfiguration.udiNumberOfCarriers < 91
        toggle SR_MulticarrierModule.xSetSingleAplMsg
        OnMouseDown: execute { SR_MulticarrierModule.udiSingleCarrierNr := 91; }
    Button (68,552 25x25), "92", colour toggle: SR_MulticarrierModule.aifVisFeedback[92].ifFeedbackConfiguration.xApplicationLoggerEntriesActive, invisible if: SR_MulticarrierModule.ifMulticarrier.ifFeedback.ifFeedbackConfiguration.udiNumberOfCarriers < 92
        toggle SR_MulticarrierModule.xSetSingleAplMsg
        OnMouseDown: execute { SR_MulticarrierModule.udiSingleCarrierNr := 92; }
    Button (108,552 25x25), "93", colour toggle: SR_MulticarrierModule.aifVisFeedback[93].ifFeedbackConfiguration.xApplicationLoggerEntriesActive, invisible if: SR_MulticarrierModule.ifMulticarrier.ifFeedback.ifFeedbackConfiguration.udiNumberOfCarriers < 93
        toggle SR_MulticarrierModule.xSetSingleAplMsg
        OnMouseDown: execute { SR_MulticarrierModule.udiSingleCarrierNr := 93; }
    Button (148,552 25x25), "94", colour toggle: SR_MulticarrierModule.aifVisFeedback[94].ifFeedbackConfiguration.xApplicationLoggerEntriesActive, invisible if: SR_MulticarrierModule.ifMulticarrier.ifFeedback.ifFeedbackConfiguration.udiNumberOfCarriers < 94
        toggle SR_MulticarrierModule.xSetSingleAplMsg
        OnMouseDown: execute { SR_MulticarrierModule.udiSingleCarrierNr := 94; }
    Button (188,552 25x25), "95", colour toggle: SR_MulticarrierModule.aifVisFeedback[95].ifFeedbackConfiguration.xApplicationLoggerEntriesActive, invisible if: SR_MulticarrierModule.ifMulticarrier.ifFeedback.ifFeedbackConfiguration.udiNumberOfCarriers < 95
        toggle SR_MulticarrierModule.xSetSingleAplMsg
        OnMouseDown: execute { SR_MulticarrierModule.udiSingleCarrierNr := 95; }
    Button (228,552 25x25), "96", colour toggle: SR_MulticarrierModule.aifVisFeedback[96].ifFeedbackConfiguration.xApplicationLoggerEntriesActive, invisible if: SR_MulticarrierModule.ifMulticarrier.ifFeedback.ifFeedbackConfiguration.udiNumberOfCarriers < 96
        toggle SR_MulticarrierModule.xSetSingleAplMsg
        OnMouseDown: execute { SR_MulticarrierModule.udiSingleCarrierNr := 96; }
    Button (268,552 25x25), "97", colour toggle: SR_MulticarrierModule.aifVisFeedback[97].ifFeedbackConfiguration.xApplicationLoggerEntriesActive, invisible if: SR_MulticarrierModule.ifMulticarrier.ifFeedback.ifFeedbackConfiguration.udiNumberOfCarriers < 97
        toggle SR_MulticarrierModule.xSetSingleAplMsg
        OnMouseDown: execute { SR_MulticarrierModule.udiSingleCarrierNr := 97; }
    Button (308,552 25x25), "98", colour toggle: SR_MulticarrierModule.aifVisFeedback[98].ifFeedbackConfiguration.xApplicationLoggerEntriesActive, invisible if: SR_MulticarrierModule.ifMulticarrier.ifFeedback.ifFeedbackConfiguration.udiNumberOfCarriers < 98
        toggle SR_MulticarrierModule.xSetSingleAplMsg
        OnMouseDown: execute { SR_MulticarrierModule.udiSingleCarrierNr := 98; }
    Button (348,552 25x25), "99", colour toggle: SR_MulticarrierModule.aifVisFeedback[99].ifFeedbackConfiguration.xApplicationLoggerEntriesActive, invisible if: SR_MulticarrierModule.ifMulticarrier.ifFeedback.ifFeedbackConfiguration.udiNumberOfCarriers < 99
        toggle SR_MulticarrierModule.xSetSingleAplMsg
        OnMouseDown: execute { SR_MulticarrierModule.udiSingleCarrierNr := 99; }
    Button (388,552 25x25), "100", colour toggle: SR_MulticarrierModule.aifVisFeedback[100].ifFeedbackConfiguration.xApplicationLoggerEntriesActive, invisible if: SR_MulticarrierModule.ifMulticarrier.ifFeedback.ifFeedbackConfiguration.udiNumberOfCarriers < 100
        toggle SR_MulticarrierModule.xSetSingleAplMsg
        OnMouseDown: execute { SR_MulticarrierModule.udiSingleCarrierNr := 100; }
    Button (28,592 25x25), "101", colour toggle: SR_MulticarrierModule.aifVisFeedback[101].ifFeedbackConfiguration.xApplicationLoggerEntriesActive, invisible if: SR_MulticarrierModule.ifMulticarrier.ifFeedback.ifFeedbackConfiguration.udiNumberOfCarriers < 101
        toggle SR_MulticarrierModule.xSetSingleAplMsg
        OnMouseDown: execute { SR_MulticarrierModule.udiSingleCarrierNr := 101; }
    Button (68,592 25x25), "102", colour toggle: SR_MulticarrierModule.aifVisFeedback[102].ifFeedbackConfiguration.xApplicationLoggerEntriesActive, invisible if: SR_MulticarrierModule.ifMulticarrier.ifFeedback.ifFeedbackConfiguration.udiNumberOfCarriers < 102
        toggle SR_MulticarrierModule.xSetSingleAplMsg
        OnMouseDown: execute { SR_MulticarrierModule.udiSingleCarrierNr := 102; }
    Button (108,592 25x25), "103", colour toggle: SR_MulticarrierModule.aifVisFeedback[103].ifFeedbackConfiguration.xApplicationLoggerEntriesActive, invisible if: SR_MulticarrierModule.ifMulticarrier.ifFeedback.ifFeedbackConfiguration.udiNumberOfCarriers < 103
        toggle SR_MulticarrierModule.xSetSingleAplMsg
        OnMouseDown: execute { SR_MulticarrierModule.udiSingleCarrierNr := 103; }
    Button (148,592 25x25), "104", colour toggle: SR_MulticarrierModule.aifVisFeedback[104].ifFeedbackConfiguration.xApplicationLoggerEntriesActive, invisible if: SR_MulticarrierModule.ifMulticarrier.ifFeedback.ifFeedbackConfiguration.udiNumberOfCarriers < 104
        toggle SR_MulticarrierModule.xSetSingleAplMsg
        OnMouseDown: execute { SR_MulticarrierModule.udiSingleCarrierNr := 104; }
    Button (188,592 25x25), "105", colour toggle: SR_MulticarrierModule.aifVisFeedback[105].ifFeedbackConfiguration.xApplicationLoggerEntriesActive, invisible if: SR_MulticarrierModule.ifMulticarrier.ifFeedback.ifFeedbackConfiguration.udiNumberOfCarriers < 105
        toggle SR_MulticarrierModule.xSetSingleAplMsg
        OnMouseDown: execute { SR_MulticarrierModule.udiSingleCarrierNr := 105; }
    Button (228,592 25x25), "106", colour toggle: SR_MulticarrierModule.aifVisFeedback[106].ifFeedbackConfiguration.xApplicationLoggerEntriesActive, invisible if: SR_MulticarrierModule.ifMulticarrier.ifFeedback.ifFeedbackConfiguration.udiNumberOfCarriers < 106
        toggle SR_MulticarrierModule.xSetSingleAplMsg
        OnMouseDown: execute { SR_MulticarrierModule.udiSingleCarrierNr := 106; }
    Button (268,592 25x25), "107", colour toggle: SR_MulticarrierModule.aifVisFeedback[107].ifFeedbackConfiguration.xApplicationLoggerEntriesActive, invisible if: SR_MulticarrierModule.ifMulticarrier.ifFeedback.ifFeedbackConfiguration.udiNumberOfCarriers < 107
        toggle SR_MulticarrierModule.xSetSingleAplMsg
        OnMouseDown: execute { SR_MulticarrierModule.udiSingleCarrierNr := 107; }
    Button (308,592 25x25), "108", colour toggle: SR_MulticarrierModule.aifVisFeedback[108].ifFeedbackConfiguration.xApplicationLoggerEntriesActive, invisible if: SR_MulticarrierModule.ifMulticarrier.ifFeedback.ifFeedbackConfiguration.udiNumberOfCarriers < 108
        toggle SR_MulticarrierModule.xSetSingleAplMsg
        OnMouseDown: execute { SR_MulticarrierModule.udiSingleCarrierNr := 108; }
    Button (348,592 25x25), "109", colour toggle: SR_MulticarrierModule.aifVisFeedback[109].ifFeedbackConfiguration.xApplicationLoggerEntriesActive, invisible if: SR_MulticarrierModule.ifMulticarrier.ifFeedback.ifFeedbackConfiguration.udiNumberOfCarriers < 109
        toggle SR_MulticarrierModule.xSetSingleAplMsg
        OnMouseDown: execute { SR_MulticarrierModule.udiSingleCarrierNr := 109; }
    Button (388,592 25x25), "110", colour toggle: SR_MulticarrierModule.aifVisFeedback[110].ifFeedbackConfiguration.xApplicationLoggerEntriesActive, invisible if: SR_MulticarrierModule.ifMulticarrier.ifFeedback.ifFeedbackConfiguration.udiNumberOfCarriers < 110
        toggle SR_MulticarrierModule.xSetSingleAplMsg
        OnMouseDown: execute { SR_MulticarrierModule.udiSingleCarrierNr := 110; }
    Button (28,632 25x25), "111", colour toggle: SR_MulticarrierModule.aifVisFeedback[111].ifFeedbackConfiguration.xApplicationLoggerEntriesActive, invisible if: SR_MulticarrierModule.ifMulticarrier.ifFeedback.ifFeedbackConfiguration.udiNumberOfCarriers < 111
        toggle SR_MulticarrierModule.xSetSingleAplMsg
        OnMouseDown: execute { SR_MulticarrierModule.udiSingleCarrierNr := 111; }
    Button (68,632 25x25), "112", colour toggle: SR_MulticarrierModule.aifVisFeedback[112].ifFeedbackConfiguration.xApplicationLoggerEntriesActive, invisible if: SR_MulticarrierModule.ifMulticarrier.ifFeedback.ifFeedbackConfiguration.udiNumberOfCarriers < 112
        toggle SR_MulticarrierModule.xSetSingleAplMsg
        OnMouseDown: execute { SR_MulticarrierModule.udiSingleCarrierNr := 112; }
    Button (108,632 25x25), "113", colour toggle: SR_MulticarrierModule.aifVisFeedback[113].ifFeedbackConfiguration.xApplicationLoggerEntriesActive, invisible if: SR_MulticarrierModule.ifMulticarrier.ifFeedback.ifFeedbackConfiguration.udiNumberOfCarriers < 113
        toggle SR_MulticarrierModule.xSetSingleAplMsg
        OnMouseDown: execute { SR_MulticarrierModule.udiSingleCarrierNr := 113; }
    Button (148,632 25x25), "114", colour toggle: SR_MulticarrierModule.aifVisFeedback[114].ifFeedbackConfiguration.xApplicationLoggerEntriesActive, invisible if: SR_MulticarrierModule.ifMulticarrier.ifFeedback.ifFeedbackConfiguration.udiNumberOfCarriers < 114
        toggle SR_MulticarrierModule.xSetSingleAplMsg
        OnMouseDown: execute { SR_MulticarrierModule.udiSingleCarrierNr := 114; }
    Button (188,632 25x25), "115", colour toggle: SR_MulticarrierModule.aifVisFeedback[115].ifFeedbackConfiguration.xApplicationLoggerEntriesActive, invisible if: SR_MulticarrierModule.ifMulticarrier.ifFeedback.ifFeedbackConfiguration.udiNumberOfCarriers < 115
        toggle SR_MulticarrierModule.xSetSingleAplMsg
        OnMouseDown: execute { SR_MulticarrierModule.udiSingleCarrierNr := 115; }
    Button (228,632 25x25), "116", colour toggle: SR_MulticarrierModule.aifVisFeedback[116].ifFeedbackConfiguration.xApplicationLoggerEntriesActive, invisible if: SR_MulticarrierModule.ifMulticarrier.ifFeedback.ifFeedbackConfiguration.udiNumberOfCarriers < 116
        toggle SR_MulticarrierModule.xSetSingleAplMsg
        OnMouseDown: execute { SR_MulticarrierModule.udiSingleCarrierNr := 116; }
    Button (268,632 25x25), "117", colour toggle: SR_MulticarrierModule.aifVisFeedback[117].ifFeedbackConfiguration.xApplicationLoggerEntriesActive, invisible if: SR_MulticarrierModule.ifMulticarrier.ifFeedback.ifFeedbackConfiguration.udiNumberOfCarriers < 117
        toggle SR_MulticarrierModule.xSetSingleAplMsg
        OnMouseDown: execute { SR_MulticarrierModule.udiSingleCarrierNr := 117; }
    Button (308,632 25x25), "118", colour toggle: SR_MulticarrierModule.aifVisFeedback[118].ifFeedbackConfiguration.xApplicationLoggerEntriesActive, invisible if: SR_MulticarrierModule.ifMulticarrier.ifFeedback.ifFeedbackConfiguration.udiNumberOfCarriers < 118
        toggle SR_MulticarrierModule.xSetSingleAplMsg
        OnMouseDown: execute { SR_MulticarrierModule.udiSingleCarrierNr := 118; }
    Button (348,632 25x25), "119", colour toggle: SR_MulticarrierModule.aifVisFeedback[119].ifFeedbackConfiguration.xApplicationLoggerEntriesActive, invisible if: SR_MulticarrierModule.ifMulticarrier.ifFeedback.ifFeedbackConfiguration.udiNumberOfCarriers < 119
        toggle SR_MulticarrierModule.xSetSingleAplMsg
        OnMouseDown: execute { SR_MulticarrierModule.udiSingleCarrierNr := 119; }
    Button (388,632 25x25), "120", colour toggle: SR_MulticarrierModule.aifVisFeedback[120].ifFeedbackConfiguration.xApplicationLoggerEntriesActive, invisible if: SR_MulticarrierModule.ifMulticarrier.ifFeedback.ifFeedbackConfiguration.udiNumberOfCarriers < 120
        toggle SR_MulticarrierModule.xSetSingleAplMsg
        OnMouseDown: execute { SR_MulticarrierModule.udiSingleCarrierNr := 120; }
    Button (28,672 25x25), "121", colour toggle: SR_MulticarrierModule.aifVisFeedback[121].ifFeedbackConfiguration.xApplicationLoggerEntriesActive, invisible if: SR_MulticarrierModule.ifMulticarrier.ifFeedback.ifFeedbackConfiguration.udiNumberOfCarriers < 121
        toggle SR_MulticarrierModule.xSetSingleAplMsg
        OnMouseDown: execute { SR_MulticarrierModule.udiSingleCarrierNr := 121; }
    Button (68,672 25x25), "122", colour toggle: SR_MulticarrierModule.aifVisFeedback[122].ifFeedbackConfiguration.xApplicationLoggerEntriesActive, invisible if: SR_MulticarrierModule.ifMulticarrier.ifFeedback.ifFeedbackConfiguration.udiNumberOfCarriers < 122
        toggle SR_MulticarrierModule.xSetSingleAplMsg
        OnMouseDown: execute { SR_MulticarrierModule.udiSingleCarrierNr := 122; }
    Button (108,672 25x25), "123", colour toggle: SR_MulticarrierModule.aifVisFeedback[123].ifFeedbackConfiguration.xApplicationLoggerEntriesActive, invisible if: SR_MulticarrierModule.ifMulticarrier.ifFeedback.ifFeedbackConfiguration.udiNumberOfCarriers < 123
        toggle SR_MulticarrierModule.xSetSingleAplMsg
        OnMouseDown: execute { SR_MulticarrierModule.udiSingleCarrierNr := 123; }
    Button (148,672 25x25), "124", colour toggle: SR_MulticarrierModule.aifVisFeedback[124].ifFeedbackConfiguration.xApplicationLoggerEntriesActive, invisible if: SR_MulticarrierModule.ifMulticarrier.ifFeedback.ifFeedbackConfiguration.udiNumberOfCarriers < 124
        toggle SR_MulticarrierModule.xSetSingleAplMsg
        OnMouseDown: execute { SR_MulticarrierModule.udiSingleCarrierNr := 124; }
    Button (388,672 25x25), "130", colour toggle: SR_MulticarrierModule.aifVisFeedback[130].ifFeedbackConfiguration.xApplicationLoggerEntriesActive, invisible if: SR_MulticarrierModule.ifMulticarrier.ifFeedback.ifFeedbackConfiguration.udiNumberOfCarriers < 130
        toggle SR_MulticarrierModule.xSetSingleAplMsg
        OnMouseDown: execute { SR_MulticarrierModule.udiSingleCarrierNr := 130; }
    Button (28,712 25x25), "131", colour toggle: SR_MulticarrierModule.aifVisFeedback[131].ifFeedbackConfiguration.xApplicationLoggerEntriesActive, invisible if: SR_MulticarrierModule.ifMulticarrier.ifFeedback.ifFeedbackConfiguration.udiNumberOfCarriers < 131
        toggle SR_MulticarrierModule.xSetSingleAplMsg
